METHOD metCreate_S_BV_5 : BOOL
(* S_BV_5*)
IF NOT S_BV_5.xIsCreated THEN
	(* Ziel						UTF8->ASCII						OBJ_NAME_BASE			BacNet Text		Textlistname									BacNet Funktion																BacNet Textlist type												TextId		*)
	S_BV_5._sObjectName		:=	fcUtfToAscii(Standard.CONCAT(	OBJ_NAME_BASE		,	fcGetBcText(	GVL_BACNET.fbBacNetParameter.metGetTextListName(enTypeOfBacNetFunktionIn := enTypeOfBacNetFunktion.Type_Automationsstation,		enTypeOfBacNetTextListIn := enTypeOfBacNetTextList.ENDING		),	'S_BV_5')));
	S_BV_5._sDescription	:= 	fcUtfToAscii(Standard.CONCAT(	OBJ_NAME_DESCRIPTION,	fcGetBcText(	GVL_BACNET.fbBacNetParameter.metGetTextListName(enTypeOfBacNetFunktionIn := enTypeOfBacNetFunktion.Type_Automationsstation,		enTypeOfBacNetTextListIn := enTypeOfBacNetTextList.DESCRIPTION	),	'S_BV_5')));
	(* Create Id from Base Id and Object Nr (Last nummber of Name *)	
	S_BV_5.Create(diInstance := TO_DINT(Standard.CONCAT(TO_STRING(dwOBJ_ID_BASE),'5')));
	(* Check if Created *)
	IF S_BV_5.xIsCreated THEN
		(* Set Group *)
		S_BV_5.setPropertyGroup(WagoTypesBacNet.eBACnetPropertyIdentifier.PROP_PRESENT_VALUE						,WagoTypesBacNet.eBACnetPropertyUpdateGroup.GROUP_CYCLIC);
		S_BV_5.setPropertyGroup(WagoTypesBacNet.eBACnetPropertyIdentifier.PROP_PRIORITY_ARRAY						,WagoTypesBacNet.eBACnetPropertyUpdateGroup.GROUP_CYCLIC);
		S_BV_5.setPropertyGroup(WagoTypesBacNet.eBACnetPropertyIdentifier.PROP_ELAPSED_ACTIVE_TIME					,WagoTypesBacNet.eBACnetPropertyUpdateGroup.GROUP_CYCLIC);
		S_BV_5.setPropertyGroup(WagoTypesBacNet.eBACnetPropertyIdentifier.PROP_DESCRIPTION							,WagoTypesBacNet.eBACnetPropertyUpdateGroup.GROUP_CYCLIC);
		S_BV_5.setPropertyGroup(WagoTypesBacNet.eBACnetPropertyIdentifier.PROP_EVENT_MESSAGE_TEXTS_CONFIG			,WagoTypesBacNet.eBACnetPropertyUpdateGroup.GROUP_CYCLIC);
		(* Set Description to Overwrite retain*)
		S_BV_5.sDescription	:= S_BV_5._sDescription;
		(* Ziel												UTF8->ASCII		BacNet Text		Textlistname									BacNet Funktion																BacNet Textlist type												TextId		*)
		S_BV_5.IEventMessageTextsConfig.sToOffNormal	:=	fcUtfToAscii(	fcGetBcText(	GVL_BACNET.fbBacNetParameter.metGetTextListName(enTypeOfBacNetFunktionIn := enTypeOfBacNetFunktion.Type_Automationsstation,		enTypeOfBacNetTextListIn := enTypeOfBacNetTextList.EVENTMESSAGE	),	'S_BV_5_ToOffNormal'	));		
		S_BV_5.IEventMessageTextsConfig.sToFault		:=	fcUtfToAscii(	fcGetBcText(	GVL_BACNET.fbBacNetParameter.metGetTextListName(enTypeOfBacNetFunktionIn := enTypeOfBacNetFunktion.Type_Automationsstation,		enTypeOfBacNetTextListIn := enTypeOfBacNetTextList.EVENTMESSAGE	),	'S_BV_5_ToFault'		));		
		S_BV_5.IEventMessageTextsConfig.sToNormal		:=	fcUtfToAscii(	fcGetBcText(	GVL_BACNET.fbBacNetParameter.metGetTextListName(enTypeOfBacNetFunktionIn := enTypeOfBacNetFunktion.Type_Automationsstation,		enTypeOfBacNetTextListIn := enTypeOfBacNetTextList.EVENTMESSAGE	),	'S_BV_5_ToNormal'		));		

		(* Ziel												UTF8->ASCII		BacNet Text		Textlistname									BacNet Funktion																BacNet Textlist type												TextId		*)	
		S_BV_5.sActiveText								:= 	fcUtfToAscii(	fcGetBcText(	GVL_BACNET.fbBacNetParameter.metGetTextListName(enTypeOfBacNetFunktionIn := enTypeOfBacNetFunktion.Type_Automationsstation,		enTypeOfBacNetTextListIn := enTypeOfBacNetTextList.PRESENTVALUE	),	'S_BV_5_ST_ACTIVE'		));
		S_BV_5.sInactiveText							:= 	fcUtfToAscii(	fcGetBcText(	GVL_BACNET.fbBacNetParameter.metGetTextListName(enTypeOfBacNetFunktionIn := enTypeOfBacNetFunktion.Type_Automationsstation,		enTypeOfBacNetTextListIn := enTypeOfBacNetTextList.PRESENTVALUE	),	'S_BV_5_ST_INACTIVE'	));	

		(* Ziel												Convert			BacNet Text		Textlistname									BacNet Funktion																	BacNet Textlist type												TextId		*)	
		S_BV_5.udiNotificationClass						:= 	TO_UDINT	(	fcGetBcText(	GVL_BACNET.fbBacNetParameter.metGetTextListName(enTypeOfBacNetFunktionIn := enTypeOfBacNetFunktion.Type_Automationsstation,		enTypeOfBacNetTextListIn := enTypeOfBacNetTextList.NC			),	'S_BV_5_NC'	));	
		S_BV_5.eNotifyType								:= 	WagoTypesBACnet.eBACnetNotifyType.NOTIFY_TYPE_ALARM;		
		S_BV_5.xAlarmValue								:= 	TO_BOOL		(	fcGetBcText(	GVL_BACNET.fbBacNetParameter.metGetTextListName(enTypeOfBacNetFunktionIn := enTypeOfBacNetFunktion.Type_Automationsstation,		enTypeOfBacNetTextListIn := enTypeOfBacNetTextList.NC			),	'S_BV_5_ALV'	));	
		
	ELSE
		S_BV_5.Delete();
	END_IF;
	(* Get Status *)
	metCreate_S_BV_5 := S_BV_5.xIsCreated;	
END_IF;
END_METHOD

METHOD metCreate_I_NC_66 : BOOL

VAR

END_VAR
(* I_NC_66*)
IF NOT I_NC_66.xIsCreated THEN
	(* Ziel						UTF8->ASCII						OBJ_NAME_BASE			BacNet Text		Textlistname									BacNet Funktion																	BacNet Textlist type												TextId		*)
	I_NC_66._sObjectName		:=	fcUtfToAscii(Standard.CONCAT(	OBJ_NAME_BASE		,	fcGetBcText(	GVL_BACNET.fbBacNetParameter.metGetTextListName(enTypeOfBacNetFunktionIn := enTypeOfBacNetFunktion.Type_Automationsstation,		enTypeOfBacNetTextListIn := enTypeOfBacNetTextList.ENDING		),	'I_NC_66')));
	I_NC_66._sDescription	:= 	fcUtfToAscii(Standard.CONCAT(	OBJ_NAME_DESCRIPTION,	fcGetBcText(	GVL_BACNET.fbBacNetParameter.metGetTextListName(enTypeOfBacNetFunktionIn := enTypeOfBacNetFunktion.Type_Automationsstation,		enTypeOfBacNetTextListIn := enTypeOfBacNetTextList.DESCRIPTION	),	'I_NC_66')));
	(* Create Id from Base Id and Object Nr (Last nummber of Name *)	
	I_NC_66.Create(diInstance := 66);
	(* Check if Created *)
	IF I_NC_66.xIsCreated THEN
		(* Set Group *)
		I_NC_66.setPropertyGroup(WagoTypesBacNet.eBACnetPropertyIdentifier.PROP_DESCRIPTION							,WagoTypesBacNet.eBACnetPropertyUpdateGroup.GROUP_CYCLIC);
		
		(* Set Ack Req *)
		I_NC_66.IAckRequired.xToOffNormal	:= TRUE;
		I_NC_66.IAckRequired.xToFault		:= TRUE;
		I_NC_66.IAckRequired.xToNormal		:= FALSE;
		
		(* Ziel												UTF8->ASCII		BacNet Text		Textlistname									BacNet Funktion																	BacNet Textlist type												TextId		*)
		I_NC_66.IEventMessageTextsConfig.sToOffNormal	:=	fcUtfToAscii(	fcGetBcText(	GVL_BACNET.fbBacNetParameter.metGetTextListName(enTypeOfBacNetFunktionIn := enTypeOfBacNetFunktion.Type_Automationsstation,		enTypeOfBacNetTextListIn := enTypeOfBacNetTextList.EVENTMESSAGE	),	'I_NC_66_ToOffNormal'	));		
		I_NC_66.IEventMessageTextsConfig.sToFault		:=	fcUtfToAscii(	fcGetBcText(	GVL_BACNET.fbBacNetParameter.metGetTextListName(enTypeOfBacNetFunktionIn := enTypeOfBacNetFunktion.Type_Automationsstation,		enTypeOfBacNetTextListIn := enTypeOfBacNetTextList.EVENTMESSAGE	),	'I_NC_66_ToFault'		));		
		I_NC_66.IEventMessageTextsConfig.sToNormal		:=	fcUtfToAscii(	fcGetBcText(	GVL_BACNET.fbBacNetParameter.metGetTextListName(enTypeOfBacNetFunktionIn := enTypeOfBacNetFunktion.Type_Automationsstation,		enTypeOfBacNetTextListIn := enTypeOfBacNetTextList.EVENTMESSAGE	),	'I_NC_66_ToNormal'		));		
		
		(* Notification Class & Type *)
		I_NC_66.udiNotificationClass					:=  66;	
		I_NC_66.eNotifyType								:= 	WagoTypesBACnet.eBACnetNotifyType.NOTIFY_TYPE_ALARM;
		(* Ziel												Convert			BacNet Text		Textlistname									BacNet Funktion																	BacNet Textlist type												TextId		*)	
		I_NC_66.IPriority.usiToOffNormal				:= 	TO_USINT(fcUtfToAscii(	fcGetBcText(	GVL_BACNET.fbBacNetParameter.metGetTextListName(enTypeOfBacNetFunktionIn := enTypeOfBacNetFunktion.Type_Automationsstation,		enTypeOfBacNetTextListIn := enTypeOfBacNetTextList.NC	),	'I_NC_66_Prio_ToOffNormal'	)));	
		I_NC_66.IPriority.usiToFault					:= 	TO_USINT(fcUtfToAscii(	fcGetBcText(	GVL_BACNET.fbBacNetParameter.metGetTextListName(enTypeOfBacNetFunktionIn := enTypeOfBacNetFunktion.Type_Automationsstation,		enTypeOfBacNetTextListIn := enTypeOfBacNetTextList.NC	),	'I_NC_66_Prio_ToFault'		)));	
		I_NC_66.IPriority.usiToNormal					:= 	TO_USINT(fcUtfToAscii(	fcGetBcText(	GVL_BACNET.fbBacNetParameter.metGetTextListName(enTypeOfBacNetFunktionIn := enTypeOfBacNetFunktion.Type_Automationsstation,		enTypeOfBacNetTextListIn := enTypeOfBacNetTextList.NC	),	'I_NC_66_Prio_ToNormal'		)));	
		
	ELSE
		I_NC_66.Delete();
	END_IF;
	(* Get Status *)
	metCreate_I_NC_66 := I_NC_66.xIsCreated;	
END_IF;
END_METHOD

METHOD metCreate_J_NC_97 : BOOL

VAR

END_VAR
(* J_NC_97*)
IF NOT J_NC_97.xIsCreated THEN
	(* Ziel						UTF8->ASCII						OBJ_NAME_BASE			BacNet Text		Textlistname									BacNet Funktion																	BacNet Textlist type												TextId		*)
	J_NC_97._sObjectName		:=	fcUtfToAscii(Standard.CONCAT(	OBJ_NAME_BASE		,	fcGetBcText(	GVL_BACNET.fbBacNetParameter.metGetTextListName(enTypeOfBacNetFunktionIn := enTypeOfBacNetFunktion.Type_Automationsstation,		enTypeOfBacNetTextListIn := enTypeOfBacNetTextList.ENDING		),	'J_NC_97')));
	J_NC_97._sDescription	:= 	fcUtfToAscii(Standard.CONCAT(	OBJ_NAME_DESCRIPTION,	fcGetBcText(	GVL_BACNET.fbBacNetParameter.metGetTextListName(enTypeOfBacNetFunktionIn := enTypeOfBacNetFunktion.Type_Automationsstation,		enTypeOfBacNetTextListIn := enTypeOfBacNetTextList.DESCRIPTION	),	'J_NC_97')));
	(* Create Id from Base Id and Object Nr (Last nummber of Name *)	
	J_NC_97.Create(diInstance := 97);
	(* Check if Created *)
	IF J_NC_97.xIsCreated THEN
		(* Set Group *)
		J_NC_97.setPropertyGroup(WagoTypesBacNet.eBACnetPropertyIdentifier.PROP_DESCRIPTION							,WagoTypesBacNet.eBACnetPropertyUpdateGroup.GROUP_CYCLIC);
		
		(* Set Ack Req *)
		J_NC_97.IAckRequired.xToOffNormal	:= FALSE;
		J_NC_97.IAckRequired.xToFault		:= TRUE;
		J_NC_97.IAckRequired.xToNormal		:= FALSE;
		
		(* Ziel												UTF8->ASCII		BacNet Text		Textlistname									BacNet Funktion																	BacNet Textlist type												TextId		*)
		J_NC_97.IEventMessageTextsConfig.sToOffNormal	:=	fcUtfToAscii(	fcGetBcText(	GVL_BACNET.fbBacNetParameter.metGetTextListName(enTypeOfBacNetFunktionIn := enTypeOfBacNetFunktion.Type_Automationsstation,		enTypeOfBacNetTextListIn := enTypeOfBacNetTextList.EVENTMESSAGE	),	'J_NC_97_ToOffNormal'	));		
		J_NC_97.IEventMessageTextsConfig.sToFault		:=	fcUtfToAscii(	fcGetBcText(	GVL_BACNET.fbBacNetParameter.metGetTextListName(enTypeOfBacNetFunktionIn := enTypeOfBacNetFunktion.Type_Automationsstation,		enTypeOfBacNetTextListIn := enTypeOfBacNetTextList.EVENTMESSAGE	),	'J_NC_97_ToFault'		));		
		J_NC_97.IEventMessageTextsConfig.sToNormal		:=	fcUtfToAscii(	fcGetBcText(	GVL_BACNET.fbBacNetParameter.metGetTextListName(enTypeOfBacNetFunktionIn := enTypeOfBacNetFunktion.Type_Automationsstation,		enTypeOfBacNetTextListIn := enTypeOfBacNetTextList.EVENTMESSAGE	),	'J_NC_97_ToNormal'		));		
		
		(* Notification Class & Type *)
		J_NC_97.udiNotificationClass					:=  97;	
		J_NC_97.eNotifyType								:= 	WagoTypesBACnet.eBACnetNotifyType.NOTIFY_TYPE_ALARM;
		(* Ziel												Convert			BacNet Text		Textlistname									BacNet Funktion																	BacNet Textlist type												TextId		*)	
		J_NC_97.IPriority.usiToOffNormal				:= 	TO_USINT(fcUtfToAscii(	fcGetBcText(	GVL_BACNET.fbBacNetParameter.metGetTextListName(enTypeOfBacNetFunktionIn := enTypeOfBacNetFunktion.Type_Automationsstation,		enTypeOfBacNetTextListIn := enTypeOfBacNetTextList.NC	),	'J_NC_97_Prio_ToOffNormal'	)));	
		J_NC_97.IPriority.usiToFault					:= 	TO_USINT(fcUtfToAscii(	fcGetBcText(	GVL_BACNET.fbBacNetParameter.metGetTextListName(enTypeOfBacNetFunktionIn := enTypeOfBacNetFunktion.Type_Automationsstation,		enTypeOfBacNetTextListIn := enTypeOfBacNetTextList.NC	),	'J_NC_97_Prio_ToFault'		)));	
		J_NC_97.IPriority.usiToNormal					:= 	TO_USINT(fcUtfToAscii(	fcGetBcText(	GVL_BACNET.fbBacNetParameter.metGetTextListName(enTypeOfBacNetFunktionIn := enTypeOfBacNetFunktion.Type_Automationsstation,		enTypeOfBacNetTextListIn := enTypeOfBacNetTextList.NC	),	'J_NC_97_Prio_ToNormal'		)));	
		
	ELSE
		J_NC_97.Delete();
	END_IF;
	(* Get Status *)
	metCreate_J_NC_97 := J_NC_97.xIsCreated;	
END_IF;
END_METHOD

METHOD metCreate_J_NC_98 : BOOL

VAR

END_VAR
(* J_NC_98*)
IF NOT J_NC_98.xIsCreated THEN
	(* Ziel						UTF8->ASCII						OBJ_NAME_BASE			BacNet Text		Textlistname									BacNet Funktion																	BacNet Textlist type												TextId		*)
	J_NC_98._sObjectName		:=	fcUtfToAscii(Standard.CONCAT(	OBJ_NAME_BASE		,	fcGetBcText(	GVL_BACNET.fbBacNetParameter.metGetTextListName(enTypeOfBacNetFunktionIn := enTypeOfBacNetFunktion.Type_Automationsstation,		enTypeOfBacNetTextListIn := enTypeOfBacNetTextList.ENDING		),	'J_NC_98')));
	J_NC_98._sDescription	:= 	fcUtfToAscii(Standard.CONCAT(	OBJ_NAME_DESCRIPTION,	fcGetBcText(	GVL_BACNET.fbBacNetParameter.metGetTextListName(enTypeOfBacNetFunktionIn := enTypeOfBacNetFunktion.Type_Automationsstation,		enTypeOfBacNetTextListIn := enTypeOfBacNetTextList.DESCRIPTION	),	'J_NC_98')));
	(* Create Id from Base Id and Object Nr (Last nummber of Name *)	
	J_NC_98.Create(diInstance := 98);
	(* Check if Created *)
	IF J_NC_98.xIsCreated THEN
		(* Set Group *)
		J_NC_98.setPropertyGroup(WagoTypesBacNet.eBACnetPropertyIdentifier.PROP_DESCRIPTION							,WagoTypesBacNet.eBACnetPropertyUpdateGroup.GROUP_CYCLIC);
		
		(* Set Ack Req *)
		J_NC_98.IAckRequired.xToOffNormal	:= TRUE;
		J_NC_98.IAckRequired.xToFault		:= TRUE;
		J_NC_98.IAckRequired.xToNormal		:= FALSE;
		
		(* Ziel												UTF8->ASCII		BacNet Text		Textlistname									BacNet Funktion																	BacNet Textlist type												TextId		*)
		J_NC_98.IEventMessageTextsConfig.sToOffNormal	:=	fcUtfToAscii(	fcGetBcText(	GVL_BACNET.fbBacNetParameter.metGetTextListName(enTypeOfBacNetFunktionIn := enTypeOfBacNetFunktion.Type_Automationsstation,		enTypeOfBacNetTextListIn := enTypeOfBacNetTextList.EVENTMESSAGE	),	'J_NC_98_ToOffNormal'	));		
		J_NC_98.IEventMessageTextsConfig.sToFault		:=	fcUtfToAscii(	fcGetBcText(	GVL_BACNET.fbBacNetParameter.metGetTextListName(enTypeOfBacNetFunktionIn := enTypeOfBacNetFunktion.Type_Automationsstation,		enTypeOfBacNetTextListIn := enTypeOfBacNetTextList.EVENTMESSAGE	),	'J_NC_98_ToFault'		));		
		J_NC_98.IEventMessageTextsConfig.sToNormal		:=	fcUtfToAscii(	fcGetBcText(	GVL_BACNET.fbBacNetParameter.metGetTextListName(enTypeOfBacNetFunktionIn := enTypeOfBacNetFunktion.Type_Automationsstation,		enTypeOfBacNetTextListIn := enTypeOfBacNetTextList.EVENTMESSAGE	),	'J_NC_98_ToNormal'		));		
		
		(* Notification Class & Type *)
		J_NC_98.udiNotificationClass					:=  98;	
		J_NC_98.eNotifyType								:= 	WagoTypesBACnet.eBACnetNotifyType.NOTIFY_TYPE_ALARM;
		(* Ziel												Convert			BacNet Text		Textlistname									BacNet Funktion																	BacNet Textlist type												TextId		*)	
		J_NC_98.IPriority.usiToOffNormal				:= 	TO_USINT(fcUtfToAscii(	fcGetBcText(	GVL_BACNET.fbBacNetParameter.metGetTextListName(enTypeOfBacNetFunktionIn := enTypeOfBacNetFunktion.Type_Automationsstation,		enTypeOfBacNetTextListIn := enTypeOfBacNetTextList.NC	),	'J_NC_98_Prio_ToOffNormal'	)));	
		J_NC_98.IPriority.usiToFault					:= 	TO_USINT(fcUtfToAscii(	fcGetBcText(	GVL_BACNET.fbBacNetParameter.metGetTextListName(enTypeOfBacNetFunktionIn := enTypeOfBacNetFunktion.Type_Automationsstation,		enTypeOfBacNetTextListIn := enTypeOfBacNetTextList.NC	),	'J_NC_98_Prio_ToFault'		)));	
		J_NC_98.IPriority.usiToNormal					:= 	TO_USINT(fcUtfToAscii(	fcGetBcText(	GVL_BACNET.fbBacNetParameter.metGetTextListName(enTypeOfBacNetFunktionIn := enTypeOfBacNetFunktion.Type_Automationsstation,		enTypeOfBacNetTextListIn := enTypeOfBacNetTextList.NC	),	'J_NC_98_Prio_ToNormal'		)));	
		
	ELSE
		J_NC_98.Delete();
	END_IF;
	(* Get Status *)
	metCreate_J_NC_98 := J_NC_98.xIsCreated;	
END_IF;
END_METHOD

METHOD metCreate_J_NC_99 : BOOL

VAR

END_VAR
(* J_NC_99*)
IF NOT J_NC_99.xIsCreated THEN
	(* Ziel						UTF8->ASCII						OBJ_NAME_BASE			BacNet Text		Textlistname									BacNet Funktion																	BacNet Textlist type												TextId		*)
	J_NC_99._sObjectName		:=	fcUtfToAscii(Standard.CONCAT(	OBJ_NAME_BASE		,	fcGetBcText(	GVL_BACNET.fbBacNetParameter.metGetTextListName(enTypeOfBacNetFunktionIn := enTypeOfBacNetFunktion.Type_Automationsstation,		enTypeOfBacNetTextListIn := enTypeOfBacNetTextList.ENDING		),	'J_NC_99')));
	J_NC_99._sDescription	:= 	fcUtfToAscii(Standard.CONCAT(	OBJ_NAME_DESCRIPTION,	fcGetBcText(	GVL_BACNET.fbBacNetParameter.metGetTextListName(enTypeOfBacNetFunktionIn := enTypeOfBacNetFunktion.Type_Automationsstation,		enTypeOfBacNetTextListIn := enTypeOfBacNetTextList.DESCRIPTION	),	'J_NC_99')));
	(* Create Id from Base Id and Object Nr (Last nummber of Name *)	
	J_NC_99.Create(diInstance := 99);
	(* Check if Created *)
	IF J_NC_99.xIsCreated THEN
		(* Set Group *)
		J_NC_99.setPropertyGroup(WagoTypesBacNet.eBACnetPropertyIdentifier.PROP_DESCRIPTION							,WagoTypesBacNet.eBACnetPropertyUpdateGroup.GROUP_CYCLIC);
		
		(* Set Ack Req *)
		J_NC_99.IAckRequired.xToOffNormal	:= TRUE;
		J_NC_99.IAckRequired.xToFault		:= TRUE;
		J_NC_99.IAckRequired.xToNormal		:= TRUE;
		
		(* Ziel												UTF8->ASCII		BacNet Text		Textlistname									BacNet Funktion																	BacNet Textlist type												TextId		*)
		J_NC_99.IEventMessageTextsConfig.sToOffNormal	:=	fcUtfToAscii(	fcGetBcText(	GVL_BACNET.fbBacNetParameter.metGetTextListName(enTypeOfBacNetFunktionIn := enTypeOfBacNetFunktion.Type_Automationsstation,		enTypeOfBacNetTextListIn := enTypeOfBacNetTextList.EVENTMESSAGE	),	'J_NC_99_ToOffNormal'	));		
		J_NC_99.IEventMessageTextsConfig.sToFault		:=	fcUtfToAscii(	fcGetBcText(	GVL_BACNET.fbBacNetParameter.metGetTextListName(enTypeOfBacNetFunktionIn := enTypeOfBacNetFunktion.Type_Automationsstation,		enTypeOfBacNetTextListIn := enTypeOfBacNetTextList.EVENTMESSAGE	),	'J_NC_99_ToFault'		));		
		J_NC_99.IEventMessageTextsConfig.sToNormal		:=	fcUtfToAscii(	fcGetBcText(	GVL_BACNET.fbBacNetParameter.metGetTextListName(enTypeOfBacNetFunktionIn := enTypeOfBacNetFunktion.Type_Automationsstation,		enTypeOfBacNetTextListIn := enTypeOfBacNetTextList.EVENTMESSAGE	),	'J_NC_99_ToNormal'		));		
		
		(* Notification Class & Type *)
		J_NC_99.udiNotificationClass					:=  99;	
		J_NC_99.eNotifyType								:= 	WagoTypesBACnet.eBACnetNotifyType.NOTIFY_TYPE_ALARM;
		(* Ziel												Convert			BacNet Text		Textlistname									BacNet Funktion																	BacNet Textlist type												TextId		*)	
		J_NC_99.IPriority.usiToOffNormal				:= 	TO_USINT(fcUtfToAscii(	fcGetBcText(	GVL_BACNET.fbBacNetParameter.metGetTextListName(enTypeOfBacNetFunktionIn := enTypeOfBacNetFunktion.Type_Automationsstation,		enTypeOfBacNetTextListIn := enTypeOfBacNetTextList.NC	),	'J_NC_99_Prio_ToOffNormal'	)));	
		J_NC_99.IPriority.usiToFault					:= 	TO_USINT(fcUtfToAscii(	fcGetBcText(	GVL_BACNET.fbBacNetParameter.metGetTextListName(enTypeOfBacNetFunktionIn := enTypeOfBacNetFunktion.Type_Automationsstation,		enTypeOfBacNetTextListIn := enTypeOfBacNetTextList.NC	),	'J_NC_99_Prio_ToFault'		)));	
		J_NC_99.IPriority.usiToNormal					:= 	TO_USINT(fcUtfToAscii(	fcGetBcText(	GVL_BACNET.fbBacNetParameter.metGetTextListName(enTypeOfBacNetFunktionIn := enTypeOfBacNetFunktion.Type_Automationsstation,		enTypeOfBacNetTextListIn := enTypeOfBacNetTextList.NC	),	'J_NC_99_Prio_ToNormal'		)));	
		
	ELSE
		J_NC_99.Delete();
	END_IF;
	(* Get Status *)
	metCreate_J_NC_99 := J_NC_99.xIsCreated;	
END_IF;
END_METHOD

METHOD metCreate_K_NC_128 : BOOL

VAR

END_VAR
(* K_NC_128*)
IF NOT K_NC_128.xIsCreated THEN
	(* Ziel						UTF8->ASCII						OBJ_NAME_BASE			BacNet Text		Textlistname									BacNet Funktion																	BacNet Textlist type												TextId		*)
	K_NC_128._sObjectName		:=	fcUtfToAscii(Standard.CONCAT(	OBJ_NAME_BASE		,	fcGetBcText(	GVL_BACNET.fbBacNetParameter.metGetTextListName(enTypeOfBacNetFunktionIn := enTypeOfBacNetFunktion.Type_Automationsstation,		enTypeOfBacNetTextListIn := enTypeOfBacNetTextList.ENDING		),	'K_NC_128')));
	K_NC_128._sDescription	:= 	fcUtfToAscii(Standard.CONCAT(	OBJ_NAME_DESCRIPTION,	fcGetBcText(	GVL_BACNET.fbBacNetParameter.metGetTextListName(enTypeOfBacNetFunktionIn := enTypeOfBacNetFunktion.Type_Automationsstation,		enTypeOfBacNetTextListIn := enTypeOfBacNetTextList.DESCRIPTION	),	'K_NC_128')));
	(* Create Id from Base Id and Object Nr (Last nummber of Name *)	
	K_NC_128.Create(diInstance := 128);
	(* Check if Created *)
	IF K_NC_128.xIsCreated THEN
		(* Set Group *)
		K_NC_128.setPropertyGroup(WagoTypesBacNet.eBACnetPropertyIdentifier.PROP_DESCRIPTION							,WagoTypesBacNet.eBACnetPropertyUpdateGroup.GROUP_CYCLIC);
		
		(* Set Ack Req *)
		K_NC_128.IAckRequired.xToOffNormal	:= FALSE;
		K_NC_128.IAckRequired.xToFault		:= FALSE;
		K_NC_128.IAckRequired.xToNormal		:= FALSE;
		
		(* Ziel												UTF8->ASCII		BacNet Text		Textlistname									BacNet Funktion																	BacNet Textlist type												TextId		*)
		K_NC_128.IEventMessageTextsConfig.sToOffNormal	:=	fcUtfToAscii(	fcGetBcText(	GVL_BACNET.fbBacNetParameter.metGetTextListName(enTypeOfBacNetFunktionIn := enTypeOfBacNetFunktion.Type_Automationsstation,		enTypeOfBacNetTextListIn := enTypeOfBacNetTextList.EVENTMESSAGE	),	'K_NC_128_ToOffNormal'	));		
		K_NC_128.IEventMessageTextsConfig.sToFault		:=	fcUtfToAscii(	fcGetBcText(	GVL_BACNET.fbBacNetParameter.metGetTextListName(enTypeOfBacNetFunktionIn := enTypeOfBacNetFunktion.Type_Automationsstation,		enTypeOfBacNetTextListIn := enTypeOfBacNetTextList.EVENTMESSAGE	),	'K_NC_128_ToFault'		));		
		K_NC_128.IEventMessageTextsConfig.sToNormal		:=	fcUtfToAscii(	fcGetBcText(	GVL_BACNET.fbBacNetParameter.metGetTextListName(enTypeOfBacNetFunktionIn := enTypeOfBacNetFunktion.Type_Automationsstation,		enTypeOfBacNetTextListIn := enTypeOfBacNetTextList.EVENTMESSAGE	),	'K_NC_128_ToNormal'		));		
		
		(* Notification Class & Type *)
		K_NC_128.udiNotificationClass					:=  128;	
		K_NC_128.eNotifyType								:= 	WagoTypesBACnet.eBACnetNotifyType.NOTIFY_TYPE_ALARM;
		(* Ziel												Convert			BacNet Text		Textlistname									BacNet Funktion																	BacNet Textlist type												TextId		*)	
		K_NC_128.IPriority.usiToOffNormal				:= 	TO_USINT(fcUtfToAscii(	fcGetBcText(	GVL_BACNET.fbBacNetParameter.metGetTextListName(enTypeOfBacNetFunktionIn := enTypeOfBacNetFunktion.Type_Automationsstation,		enTypeOfBacNetTextListIn := enTypeOfBacNetTextList.NC	),	'K_NC_128_Prio_ToOffNormal'	)));	
		K_NC_128.IPriority.usiToFault					:= 	TO_USINT(fcUtfToAscii(	fcGetBcText(	GVL_BACNET.fbBacNetParameter.metGetTextListName(enTypeOfBacNetFunktionIn := enTypeOfBacNetFunktion.Type_Automationsstation,		enTypeOfBacNetTextListIn := enTypeOfBacNetTextList.NC	),	'K_NC_128_Prio_ToFault'		)));	
		K_NC_128.IPriority.usiToNormal					:= 	TO_USINT(fcUtfToAscii(	fcGetBcText(	GVL_BACNET.fbBacNetParameter.metGetTextListName(enTypeOfBacNetFunktionIn := enTypeOfBacNetFunktion.Type_Automationsstation,		enTypeOfBacNetTextListIn := enTypeOfBacNetTextList.NC	),	'K_NC_128_Prio_ToNormal'		)));	
		
	ELSE
		K_NC_128.Delete();
	END_IF;
	(* Get Status *)
	metCreate_K_NC_128 := K_NC_128.xIsCreated;	
END_IF;
END_METHOD

METHOD metCreate_H_NC_35 : BOOL

VAR

END_VAR
(* H_NC_35*)
IF NOT H_NC_35.xIsCreated THEN
	(* Ziel						UTF8->ASCII						OBJ_NAME_BASE			BacNet Text		Textlistname									BacNet Funktion																	BacNet Textlist type												TextId		*)
	H_NC_35._sObjectName		:=	fcUtfToAscii(Standard.CONCAT(	OBJ_NAME_BASE		,	fcGetBcText(	GVL_BACNET.fbBacNetParameter.metGetTextListName(enTypeOfBacNetFunktionIn := enTypeOfBacNetFunktion.Type_Automationsstation,		enTypeOfBacNetTextListIn := enTypeOfBacNetTextList.ENDING		),	'H_NC_35')));
	H_NC_35._sDescription	:= 	fcUtfToAscii(Standard.CONCAT(	OBJ_NAME_DESCRIPTION,	fcGetBcText(	GVL_BACNET.fbBacNetParameter.metGetTextListName(enTypeOfBacNetFunktionIn := enTypeOfBacNetFunktion.Type_Automationsstation,		enTypeOfBacNetTextListIn := enTypeOfBacNetTextList.DESCRIPTION	),	'H_NC_35')));
	(* Create Id from Base Id and Object Nr (Last nummber of Name *)	
	H_NC_35.Create(diInstance := 35);
	(* Check if Created *)
	IF H_NC_35.xIsCreated THEN
		(* Set Group *)
		H_NC_35.setPropertyGroup(WagoTypesBacNet.eBACnetPropertyIdentifier.PROP_DESCRIPTION							,WagoTypesBacNet.eBACnetPropertyUpdateGroup.GROUP_CYCLIC);
		
		(* Set Ack Req *)
		H_NC_35.IAckRequired.xToOffNormal	:= TRUE;
		H_NC_35.IAckRequired.xToFault		:= TRUE;
		H_NC_35.IAckRequired.xToNormal		:= TRUE;
		
		(* Ziel												UTF8->ASCII		BacNet Text		Textlistname									BacNet Funktion																	BacNet Textlist type												TextId		*)
		H_NC_35.IEventMessageTextsConfig.sToOffNormal	:=	fcUtfToAscii(	fcGetBcText(	GVL_BACNET.fbBacNetParameter.metGetTextListName(enTypeOfBacNetFunktionIn := enTypeOfBacNetFunktion.Type_Automationsstation,		enTypeOfBacNetTextListIn := enTypeOfBacNetTextList.EVENTMESSAGE	),	'H_NC_35_ToOffNormal'	));		
		H_NC_35.IEventMessageTextsConfig.sToFault		:=	fcUtfToAscii(	fcGetBcText(	GVL_BACNET.fbBacNetParameter.metGetTextListName(enTypeOfBacNetFunktionIn := enTypeOfBacNetFunktion.Type_Automationsstation,		enTypeOfBacNetTextListIn := enTypeOfBacNetTextList.EVENTMESSAGE	),	'H_NC_35_ToFault'		));		
		H_NC_35.IEventMessageTextsConfig.sToNormal		:=	fcUtfToAscii(	fcGetBcText(	GVL_BACNET.fbBacNetParameter.metGetTextListName(enTypeOfBacNetFunktionIn := enTypeOfBacNetFunktion.Type_Automationsstation,		enTypeOfBacNetTextListIn := enTypeOfBacNetTextList.EVENTMESSAGE	),	'H_NC_35_ToNormal'		));		
		
		(* Notification Class & Type *)
		H_NC_35.udiNotificationClass					:=  35;	
		H_NC_35.eNotifyType								:= 	WagoTypesBACnet.eBACnetNotifyType.NOTIFY_TYPE_ALARM;
		(* Ziel												Convert			BacNet Text		Textlistname									BacNet Funktion																	BacNet Textlist type												TextId		*)	
		H_NC_35.IPriority.usiToOffNormal				:= 	TO_USINT(fcUtfToAscii(	fcGetBcText(	GVL_BACNET.fbBacNetParameter.metGetTextListName(enTypeOfBacNetFunktionIn := enTypeOfBacNetFunktion.Type_Automationsstation,		enTypeOfBacNetTextListIn := enTypeOfBacNetTextList.NC	),	'H_NC_35_Prio_ToOffNormal'	)));	
		H_NC_35.IPriority.usiToFault					:= 	TO_USINT(fcUtfToAscii(	fcGetBcText(	GVL_BACNET.fbBacNetParameter.metGetTextListName(enTypeOfBacNetFunktionIn := enTypeOfBacNetFunktion.Type_Automationsstation,		enTypeOfBacNetTextListIn := enTypeOfBacNetTextList.NC	),	'H_NC_35_Prio_ToFault'		)));	
		H_NC_35.IPriority.usiToNormal					:= 	TO_USINT(fcUtfToAscii(	fcGetBcText(	GVL_BACNET.fbBacNetParameter.metGetTextListName(enTypeOfBacNetFunktionIn := enTypeOfBacNetFunktion.Type_Automationsstation,		enTypeOfBacNetTextListIn := enTypeOfBacNetTextList.NC	),	'H_NC_35_Prio_ToNormal'		)));	
		
	ELSE
		H_NC_35.Delete();
	END_IF;
	(* Get Status *)
	metCreate_H_NC_35 := H_NC_35.xIsCreated;	
END_IF;
END_METHOD

METHOD metCreate_I_NC_64 : BOOL

VAR

END_VAR
(* I_NC_64*)
IF NOT I_NC_64.xIsCreated THEN
	(* Ziel						UTF8->ASCII						OBJ_NAME_BASE			BacNet Text		Textlistname									BacNet Funktion																	BacNet Textlist type												TextId		*)
	I_NC_64._sObjectName		:=	fcUtfToAscii(Standard.CONCAT(	OBJ_NAME_BASE		,	fcGetBcText(	GVL_BACNET.fbBacNetParameter.metGetTextListName(enTypeOfBacNetFunktionIn := enTypeOfBacNetFunktion.Type_Automationsstation,		enTypeOfBacNetTextListIn := enTypeOfBacNetTextList.ENDING		),	'I_NC_64')));
	I_NC_64._sDescription	:= 	fcUtfToAscii(Standard.CONCAT(	OBJ_NAME_DESCRIPTION,	fcGetBcText(	GVL_BACNET.fbBacNetParameter.metGetTextListName(enTypeOfBacNetFunktionIn := enTypeOfBacNetFunktion.Type_Automationsstation,		enTypeOfBacNetTextListIn := enTypeOfBacNetTextList.DESCRIPTION	),	'I_NC_64')));
	(* Create Id from Base Id and Object Nr (Last nummber of Name *)	
	I_NC_64.Create(diInstance := 64);
	(* Check if Created *)
	IF I_NC_64.xIsCreated THEN
		(* Set Group *)
		I_NC_64.setPropertyGroup(WagoTypesBacNet.eBACnetPropertyIdentifier.PROP_DESCRIPTION							,WagoTypesBacNet.eBACnetPropertyUpdateGroup.GROUP_CYCLIC);
		
		(* Set Ack Req *)
		I_NC_64.IAckRequired.xToOffNormal	:= FALSE;
		I_NC_64.IAckRequired.xToFault		:= FALSE;
		I_NC_64.IAckRequired.xToNormal		:= FALSE;
		
		(* Ziel												UTF8->ASCII		BacNet Text		Textlistname									BacNet Funktion																	BacNet Textlist type												TextId		*)
		I_NC_64.IEventMessageTextsConfig.sToOffNormal	:=	fcUtfToAscii(	fcGetBcText(	GVL_BACNET.fbBacNetParameter.metGetTextListName(enTypeOfBacNetFunktionIn := enTypeOfBacNetFunktion.Type_Automationsstation,		enTypeOfBacNetTextListIn := enTypeOfBacNetTextList.EVENTMESSAGE	),	'I_NC_64_ToOffNormal'	));		
		I_NC_64.IEventMessageTextsConfig.sToFault		:=	fcUtfToAscii(	fcGetBcText(	GVL_BACNET.fbBacNetParameter.metGetTextListName(enTypeOfBacNetFunktionIn := enTypeOfBacNetFunktion.Type_Automationsstation,		enTypeOfBacNetTextListIn := enTypeOfBacNetTextList.EVENTMESSAGE	),	'I_NC_64_ToFault'		));		
		I_NC_64.IEventMessageTextsConfig.sToNormal		:=	fcUtfToAscii(	fcGetBcText(	GVL_BACNET.fbBacNetParameter.metGetTextListName(enTypeOfBacNetFunktionIn := enTypeOfBacNetFunktion.Type_Automationsstation,		enTypeOfBacNetTextListIn := enTypeOfBacNetTextList.EVENTMESSAGE	),	'I_NC_64_ToNormal'		));		
		
		(* Notification Class & Type *)
		I_NC_64.udiNotificationClass					:=  64;	
		I_NC_64.eNotifyType								:= 	WagoTypesBACnet.eBACnetNotifyType.NOTIFY_TYPE_ALARM;
		(* Ziel												Convert			BacNet Text		Textlistname									BacNet Funktion																	BacNet Textlist type												TextId		*)	
		I_NC_64.IPriority.usiToOffNormal				:= 	TO_USINT(fcUtfToAscii(	fcGetBcText(	GVL_BACNET.fbBacNetParameter.metGetTextListName(enTypeOfBacNetFunktionIn := enTypeOfBacNetFunktion.Type_Automationsstation,		enTypeOfBacNetTextListIn := enTypeOfBacNetTextList.NC	),	'I_NC_64_Prio_ToOffNormal'	)));	
		I_NC_64.IPriority.usiToFault					:= 	TO_USINT(fcUtfToAscii(	fcGetBcText(	GVL_BACNET.fbBacNetParameter.metGetTextListName(enTypeOfBacNetFunktionIn := enTypeOfBacNetFunktion.Type_Automationsstation,		enTypeOfBacNetTextListIn := enTypeOfBacNetTextList.NC	),	'I_NC_64_Prio_ToFault'		)));	
		I_NC_64.IPriority.usiToNormal					:= 	TO_USINT(fcUtfToAscii(	fcGetBcText(	GVL_BACNET.fbBacNetParameter.metGetTextListName(enTypeOfBacNetFunktionIn := enTypeOfBacNetFunktion.Type_Automationsstation,		enTypeOfBacNetTextListIn := enTypeOfBacNetTextList.NC	),	'I_NC_64_Prio_ToNormal'		)));	
		
	ELSE
		I_NC_64.Delete();
	END_IF;
	(* Get Status *)
	metCreate_I_NC_64 := I_NC_64.xIsCreated;	
END_IF;
END_METHOD

METHOD metCreate_I_NC_67 : BOOL

VAR

END_VAR
(* I_NC_67*)
IF NOT I_NC_67.xIsCreated THEN
	(* Ziel						UTF8->ASCII						OBJ_NAME_BASE			BacNet Text		Textlistname									BacNet Funktion																	BacNet Textlist type												TextId		*)
	I_NC_67._sObjectName		:=	fcUtfToAscii(Standard.CONCAT(	OBJ_NAME_BASE		,	fcGetBcText(	GVL_BACNET.fbBacNetParameter.metGetTextListName(enTypeOfBacNetFunktionIn := enTypeOfBacNetFunktion.Type_Automationsstation,		enTypeOfBacNetTextListIn := enTypeOfBacNetTextList.ENDING		),	'I_NC_67')));
	I_NC_67._sDescription	:= 	fcUtfToAscii(Standard.CONCAT(	OBJ_NAME_DESCRIPTION,	fcGetBcText(	GVL_BACNET.fbBacNetParameter.metGetTextListName(enTypeOfBacNetFunktionIn := enTypeOfBacNetFunktion.Type_Automationsstation,		enTypeOfBacNetTextListIn := enTypeOfBacNetTextList.DESCRIPTION	),	'I_NC_67')));
	(* Create Id from Base Id and Object Nr (Last nummber of Name *)	
	I_NC_67.Create(diInstance := 67);
	(* Check if Created *)
	IF I_NC_67.xIsCreated THEN
		(* Set Group *)
		I_NC_67.setPropertyGroup(WagoTypesBacNet.eBACnetPropertyIdentifier.PROP_DESCRIPTION							,WagoTypesBacNet.eBACnetPropertyUpdateGroup.GROUP_CYCLIC);
		
		(* Set Ack Req *)
		I_NC_67.IAckRequired.xToOffNormal	:= TRUE;
		I_NC_67.IAckRequired.xToFault		:= TRUE;
		I_NC_67.IAckRequired.xToNormal		:= TRUE;
		
		(* Ziel												UTF8->ASCII		BacNet Text		Textlistname									BacNet Funktion																	BacNet Textlist type												TextId		*)
		I_NC_67.IEventMessageTextsConfig.sToOffNormal	:=	fcUtfToAscii(	fcGetBcText(	GVL_BACNET.fbBacNetParameter.metGetTextListName(enTypeOfBacNetFunktionIn := enTypeOfBacNetFunktion.Type_Automationsstation,		enTypeOfBacNetTextListIn := enTypeOfBacNetTextList.EVENTMESSAGE	),	'I_NC_67_ToOffNormal'	));		
		I_NC_67.IEventMessageTextsConfig.sToFault		:=	fcUtfToAscii(	fcGetBcText(	GVL_BACNET.fbBacNetParameter.metGetTextListName(enTypeOfBacNetFunktionIn := enTypeOfBacNetFunktion.Type_Automationsstation,		enTypeOfBacNetTextListIn := enTypeOfBacNetTextList.EVENTMESSAGE	),	'I_NC_67_ToFault'		));		
		I_NC_67.IEventMessageTextsConfig.sToNormal		:=	fcUtfToAscii(	fcGetBcText(	GVL_BACNET.fbBacNetParameter.metGetTextListName(enTypeOfBacNetFunktionIn := enTypeOfBacNetFunktion.Type_Automationsstation,		enTypeOfBacNetTextListIn := enTypeOfBacNetTextList.EVENTMESSAGE	),	'I_NC_67_ToNormal'		));		
		
		(* Notification Class & Type *)
		I_NC_67.udiNotificationClass					:=  67;	
		I_NC_67.eNotifyType								:= 	WagoTypesBACnet.eBACnetNotifyType.NOTIFY_TYPE_ALARM;
		(* Ziel												Convert			BacNet Text		Textlistname									BacNet Funktion																	BacNet Textlist type												TextId		*)	
		I_NC_67.IPriority.usiToOffNormal				:= 	TO_USINT(fcUtfToAscii(	fcGetBcText(	GVL_BACNET.fbBacNetParameter.metGetTextListName(enTypeOfBacNetFunktionIn := enTypeOfBacNetFunktion.Type_Automationsstation,		enTypeOfBacNetTextListIn := enTypeOfBacNetTextList.NC	),	'I_NC_67_Prio_ToOffNormal'	)));	
		I_NC_67.IPriority.usiToFault					:= 	TO_USINT(fcUtfToAscii(	fcGetBcText(	GVL_BACNET.fbBacNetParameter.metGetTextListName(enTypeOfBacNetFunktionIn := enTypeOfBacNetFunktion.Type_Automationsstation,		enTypeOfBacNetTextListIn := enTypeOfBacNetTextList.NC	),	'I_NC_67_Prio_ToFault'		)));	
		I_NC_67.IPriority.usiToNormal					:= 	TO_USINT(fcUtfToAscii(	fcGetBcText(	GVL_BACNET.fbBacNetParameter.metGetTextListName(enTypeOfBacNetFunktionIn := enTypeOfBacNetFunktion.Type_Automationsstation,		enTypeOfBacNetTextListIn := enTypeOfBacNetTextList.NC	),	'I_NC_67_Prio_ToNormal'		)));	
		
	ELSE
		I_NC_67.Delete();
	END_IF;
	(* Get Status *)
	metCreate_I_NC_67 := I_NC_67.xIsCreated;	
END_IF;
END_METHOD

METHOD metCreate_J_NC_96 : BOOL

VAR

END_VAR
(* J_NC_96*)
IF NOT J_NC_96.xIsCreated THEN
	(* Ziel						UTF8->ASCII						OBJ_NAME_BASE			BacNet Text		Textlistname									BacNet Funktion																	BacNet Textlist type												TextId		*)
	J_NC_96._sObjectName		:=	fcUtfToAscii(Standard.CONCAT(	OBJ_NAME_BASE		,	fcGetBcText(	GVL_BACNET.fbBacNetParameter.metGetTextListName(enTypeOfBacNetFunktionIn := enTypeOfBacNetFunktion.Type_Automationsstation,		enTypeOfBacNetTextListIn := enTypeOfBacNetTextList.ENDING		),	'J_NC_96')));
	J_NC_96._sDescription	:= 	fcUtfToAscii(Standard.CONCAT(	OBJ_NAME_DESCRIPTION,	fcGetBcText(	GVL_BACNET.fbBacNetParameter.metGetTextListName(enTypeOfBacNetFunktionIn := enTypeOfBacNetFunktion.Type_Automationsstation,		enTypeOfBacNetTextListIn := enTypeOfBacNetTextList.DESCRIPTION	),	'J_NC_96')));
	(* Create Id from Base Id and Object Nr (Last nummber of Name *)	
	J_NC_96.Create(diInstance := 96);
	(* Check if Created *)
	IF J_NC_96.xIsCreated THEN
		(* Set Group *)
		J_NC_96.setPropertyGroup(WagoTypesBacNet.eBACnetPropertyIdentifier.PROP_DESCRIPTION							,WagoTypesBacNet.eBACnetPropertyUpdateGroup.GROUP_CYCLIC);
		
		(* Set Ack Req *)
		J_NC_96.IAckRequired.xToOffNormal	:= FALSE;
		J_NC_96.IAckRequired.xToFault		:= FALSE;
		J_NC_96.IAckRequired.xToNormal		:= FALSE;
		
		(* Ziel												UTF8->ASCII		BacNet Text		Textlistname									BacNet Funktion																	BacNet Textlist type												TextId		*)
		J_NC_96.IEventMessageTextsConfig.sToOffNormal	:=	fcUtfToAscii(	fcGetBcText(	GVL_BACNET.fbBacNetParameter.metGetTextListName(enTypeOfBacNetFunktionIn := enTypeOfBacNetFunktion.Type_Automationsstation,		enTypeOfBacNetTextListIn := enTypeOfBacNetTextList.EVENTMESSAGE	),	'J_NC_96_ToOffNormal'	));		
		J_NC_96.IEventMessageTextsConfig.sToFault		:=	fcUtfToAscii(	fcGetBcText(	GVL_BACNET.fbBacNetParameter.metGetTextListName(enTypeOfBacNetFunktionIn := enTypeOfBacNetFunktion.Type_Automationsstation,		enTypeOfBacNetTextListIn := enTypeOfBacNetTextList.EVENTMESSAGE	),	'J_NC_96_ToFault'		));		
		J_NC_96.IEventMessageTextsConfig.sToNormal		:=	fcUtfToAscii(	fcGetBcText(	GVL_BACNET.fbBacNetParameter.metGetTextListName(enTypeOfBacNetFunktionIn := enTypeOfBacNetFunktion.Type_Automationsstation,		enTypeOfBacNetTextListIn := enTypeOfBacNetTextList.EVENTMESSAGE	),	'J_NC_96_ToNormal'		));		
		
		(* Notification Class & Type *)
		J_NC_96.udiNotificationClass					:=  96;	
		J_NC_96.eNotifyType								:= 	WagoTypesBACnet.eBACnetNotifyType.NOTIFY_TYPE_ALARM;
		(* Ziel												Convert			BacNet Text		Textlistname									BacNet Funktion																	BacNet Textlist type												TextId		*)	
		J_NC_96.IPriority.usiToOffNormal				:= 	TO_USINT(fcUtfToAscii(	fcGetBcText(	GVL_BACNET.fbBacNetParameter.metGetTextListName(enTypeOfBacNetFunktionIn := enTypeOfBacNetFunktion.Type_Automationsstation,		enTypeOfBacNetTextListIn := enTypeOfBacNetTextList.NC	),	'J_NC_96_Prio_ToOffNormal'	)));	
		J_NC_96.IPriority.usiToFault					:= 	TO_USINT(fcUtfToAscii(	fcGetBcText(	GVL_BACNET.fbBacNetParameter.metGetTextListName(enTypeOfBacNetFunktionIn := enTypeOfBacNetFunktion.Type_Automationsstation,		enTypeOfBacNetTextListIn := enTypeOfBacNetTextList.NC	),	'J_NC_96_Prio_ToFault'		)));	
		J_NC_96.IPriority.usiToNormal					:= 	TO_USINT(fcUtfToAscii(	fcGetBcText(	GVL_BACNET.fbBacNetParameter.metGetTextListName(enTypeOfBacNetFunktionIn := enTypeOfBacNetFunktion.Type_Automationsstation,		enTypeOfBacNetTextListIn := enTypeOfBacNetTextList.NC	),	'J_NC_96_Prio_ToNormal'		)));	
		
	ELSE
		J_NC_96.Delete();
	END_IF;
	(* Get Status *)
	metCreate_J_NC_96 := J_NC_96.xIsCreated;	
END_IF;
END_METHOD

METHOD metCreate_K_NC_129 : BOOL

VAR

END_VAR
(* K_NC_129*)
IF NOT K_NC_129.xIsCreated THEN
	(* Ziel						UTF8->ASCII						OBJ_NAME_BASE			BacNet Text		Textlistname									BacNet Funktion																	BacNet Textlist type												TextId		*)
	K_NC_129._sObjectName		:=	fcUtfToAscii(Standard.CONCAT(	OBJ_NAME_BASE		,	fcGetBcText(	GVL_BACNET.fbBacNetParameter.metGetTextListName(enTypeOfBacNetFunktionIn := enTypeOfBacNetFunktion.Type_Automationsstation,		enTypeOfBacNetTextListIn := enTypeOfBacNetTextList.ENDING		),	'K_NC_129')));
	K_NC_129._sDescription	:= 	fcUtfToAscii(Standard.CONCAT(	OBJ_NAME_DESCRIPTION,	fcGetBcText(	GVL_BACNET.fbBacNetParameter.metGetTextListName(enTypeOfBacNetFunktionIn := enTypeOfBacNetFunktion.Type_Automationsstation,		enTypeOfBacNetTextListIn := enTypeOfBacNetTextList.DESCRIPTION	),	'K_NC_129')));
	(* Create Id from Base Id and Object Nr (Last nummber of Name *)	
	K_NC_129.Create(diInstance := 129);
	(* Check if Created *)
	IF K_NC_129.xIsCreated THEN
		(* Set Group *)
		K_NC_129.setPropertyGroup(WagoTypesBacNet.eBACnetPropertyIdentifier.PROP_DESCRIPTION							,WagoTypesBacNet.eBACnetPropertyUpdateGroup.GROUP_CYCLIC);
		
		(* Set Ack Req *)
		K_NC_129.IAckRequired.xToOffNormal	:= FALSE;
		K_NC_129.IAckRequired.xToFault		:= TRUE;
		K_NC_129.IAckRequired.xToNormal		:= FALSE;
		
		(* Ziel												UTF8->ASCII		BacNet Text		Textlistname									BacNet Funktion																	BacNet Textlist type												TextId		*)
		K_NC_129.IEventMessageTextsConfig.sToOffNormal	:=	fcUtfToAscii(	fcGetBcText(	GVL_BACNET.fbBacNetParameter.metGetTextListName(enTypeOfBacNetFunktionIn := enTypeOfBacNetFunktion.Type_Automationsstation,		enTypeOfBacNetTextListIn := enTypeOfBacNetTextList.EVENTMESSAGE	),	'K_NC_129_ToOffNormal'	));		
		K_NC_129.IEventMessageTextsConfig.sToFault		:=	fcUtfToAscii(	fcGetBcText(	GVL_BACNET.fbBacNetParameter.metGetTextListName(enTypeOfBacNetFunktionIn := enTypeOfBacNetFunktion.Type_Automationsstation,		enTypeOfBacNetTextListIn := enTypeOfBacNetTextList.EVENTMESSAGE	),	'K_NC_129_ToFault'		));		
		K_NC_129.IEventMessageTextsConfig.sToNormal		:=	fcUtfToAscii(	fcGetBcText(	GVL_BACNET.fbBacNetParameter.metGetTextListName(enTypeOfBacNetFunktionIn := enTypeOfBacNetFunktion.Type_Automationsstation,		enTypeOfBacNetTextListIn := enTypeOfBacNetTextList.EVENTMESSAGE	),	'K_NC_129_ToNormal'		));		
		
		(* Notification Class & Type *)
		K_NC_129.udiNotificationClass					:=  129;	
		K_NC_129.eNotifyType								:= 	WagoTypesBACnet.eBACnetNotifyType.NOTIFY_TYPE_ALARM;
		(* Ziel												Convert			BacNet Text		Textlistname									BacNet Funktion																	BacNet Textlist type												TextId		*)	
		K_NC_129.IPriority.usiToOffNormal				:= 	TO_USINT(fcUtfToAscii(	fcGetBcText(	GVL_BACNET.fbBacNetParameter.metGetTextListName(enTypeOfBacNetFunktionIn := enTypeOfBacNetFunktion.Type_Automationsstation,		enTypeOfBacNetTextListIn := enTypeOfBacNetTextList.NC	),	'K_NC_129_Prio_ToOffNormal'	)));	
		K_NC_129.IPriority.usiToFault					:= 	TO_USINT(fcUtfToAscii(	fcGetBcText(	GVL_BACNET.fbBacNetParameter.metGetTextListName(enTypeOfBacNetFunktionIn := enTypeOfBacNetFunktion.Type_Automationsstation,		enTypeOfBacNetTextListIn := enTypeOfBacNetTextList.NC	),	'K_NC_129_Prio_ToFault'		)));	
		K_NC_129.IPriority.usiToNormal					:= 	TO_USINT(fcUtfToAscii(	fcGetBcText(	GVL_BACNET.fbBacNetParameter.metGetTextListName(enTypeOfBacNetFunktionIn := enTypeOfBacNetFunktion.Type_Automationsstation,		enTypeOfBacNetTextListIn := enTypeOfBacNetTextList.NC	),	'K_NC_129_Prio_ToNormal'		)));	
		
	ELSE
		K_NC_129.Delete();
	END_IF;
	(* Get Status *)
	metCreate_K_NC_129 := K_NC_129.xIsCreated;	
END_IF;
END_METHOD

METHOD metCreate_K_NC_130 : BOOL

VAR

END_VAR
(* K_NC_130*)
IF NOT K_NC_130.xIsCreated THEN
	(* Ziel						UTF8->ASCII						OBJ_NAME_BASE			BacNet Text		Textlistname									BacNet Funktion																	BacNet Textlist type												TextId		*)
	K_NC_130._sObjectName		:=	fcUtfToAscii(Standard.CONCAT(	OBJ_NAME_BASE		,	fcGetBcText(	GVL_BACNET.fbBacNetParameter.metGetTextListName(enTypeOfBacNetFunktionIn := enTypeOfBacNetFunktion.Type_Automationsstation,		enTypeOfBacNetTextListIn := enTypeOfBacNetTextList.ENDING		),	'K_NC_130')));
	K_NC_130._sDescription	:= 	fcUtfToAscii(Standard.CONCAT(	OBJ_NAME_DESCRIPTION,	fcGetBcText(	GVL_BACNET.fbBacNetParameter.metGetTextListName(enTypeOfBacNetFunktionIn := enTypeOfBacNetFunktion.Type_Automationsstation,		enTypeOfBacNetTextListIn := enTypeOfBacNetTextList.DESCRIPTION	),	'K_NC_130')));
	(* Create Id from Base Id and Object Nr (Last nummber of Name *)	
	K_NC_130.Create(diInstance := 130);
	(* Check if Created *)
	IF K_NC_130.xIsCreated THEN
		(* Set Group *)
		K_NC_130.setPropertyGroup(WagoTypesBacNet.eBACnetPropertyIdentifier.PROP_DESCRIPTION							,WagoTypesBacNet.eBACnetPropertyUpdateGroup.GROUP_CYCLIC);
		
		(* Set Ack Req *)
		K_NC_130.IAckRequired.xToOffNormal	:= TRUE;
		K_NC_130.IAckRequired.xToFault		:= TRUE;
		K_NC_130.IAckRequired.xToNormal		:= FALSE;
		
		(* Ziel												UTF8->ASCII		BacNet Text		Textlistname									BacNet Funktion																	BacNet Textlist type												TextId		*)
		K_NC_130.IEventMessageTextsConfig.sToOffNormal	:=	fcUtfToAscii(	fcGetBcText(	GVL_BACNET.fbBacNetParameter.metGetTextListName(enTypeOfBacNetFunktionIn := enTypeOfBacNetFunktion.Type_Automationsstation,		enTypeOfBacNetTextListIn := enTypeOfBacNetTextList.EVENTMESSAGE	),	'K_NC_130_ToOffNormal'	));		
		K_NC_130.IEventMessageTextsConfig.sToFault		:=	fcUtfToAscii(	fcGetBcText(	GVL_BACNET.fbBacNetParameter.metGetTextListName(enTypeOfBacNetFunktionIn := enTypeOfBacNetFunktion.Type_Automationsstation,		enTypeOfBacNetTextListIn := enTypeOfBacNetTextList.EVENTMESSAGE	),	'K_NC_130_ToFault'		));		
		K_NC_130.IEventMessageTextsConfig.sToNormal		:=	fcUtfToAscii(	fcGetBcText(	GVL_BACNET.fbBacNetParameter.metGetTextListName(enTypeOfBacNetFunktionIn := enTypeOfBacNetFunktion.Type_Automationsstation,		enTypeOfBacNetTextListIn := enTypeOfBacNetTextList.EVENTMESSAGE	),	'K_NC_130_ToNormal'		));		
		
		(* Notification Class & Type *)
		K_NC_130.udiNotificationClass					:=  130;	
		K_NC_130.eNotifyType								:= 	WagoTypesBACnet.eBACnetNotifyType.NOTIFY_TYPE_ALARM;
		(* Ziel												Convert			BacNet Text		Textlistname									BacNet Funktion																	BacNet Textlist type												TextId		*)	
		K_NC_130.IPriority.usiToOffNormal				:= 	TO_USINT(fcUtfToAscii(	fcGetBcText(	GVL_BACNET.fbBacNetParameter.metGetTextListName(enTypeOfBacNetFunktionIn := enTypeOfBacNetFunktion.Type_Automationsstation,		enTypeOfBacNetTextListIn := enTypeOfBacNetTextList.NC	),	'K_NC_130_Prio_ToOffNormal'	)));	
		K_NC_130.IPriority.usiToFault					:= 	TO_USINT(fcUtfToAscii(	fcGetBcText(	GVL_BACNET.fbBacNetParameter.metGetTextListName(enTypeOfBacNetFunktionIn := enTypeOfBacNetFunktion.Type_Automationsstation,		enTypeOfBacNetTextListIn := enTypeOfBacNetTextList.NC	),	'K_NC_130_Prio_ToFault'		)));	
		K_NC_130.IPriority.usiToNormal					:= 	TO_USINT(fcUtfToAscii(	fcGetBcText(	GVL_BACNET.fbBacNetParameter.metGetTextListName(enTypeOfBacNetFunktionIn := enTypeOfBacNetFunktion.Type_Automationsstation,		enTypeOfBacNetTextListIn := enTypeOfBacNetTextList.NC	),	'K_NC_130_Prio_ToNormal'		)));	
		
	ELSE
		K_NC_130.Delete();
	END_IF;
	(* Get Status *)
	metCreate_K_NC_130 := K_NC_130.xIsCreated;	
END_IF;
END_METHOD

METHOD metCreate_K_NC_131 : BOOL

VAR

END_VAR
(* K_NC_131*)
IF NOT K_NC_131.xIsCreated THEN
	(* Ziel						UTF8->ASCII						OBJ_NAME_BASE			BacNet Text		Textlistname									BacNet Funktion																	BacNet Textlist type												TextId		*)
	K_NC_131._sObjectName		:=	fcUtfToAscii(Standard.CONCAT(	OBJ_NAME_BASE		,	fcGetBcText(	GVL_BACNET.fbBacNetParameter.metGetTextListName(enTypeOfBacNetFunktionIn := enTypeOfBacNetFunktion.Type_Automationsstation,		enTypeOfBacNetTextListIn := enTypeOfBacNetTextList.ENDING		),	'K_NC_131')));
	K_NC_131._sDescription	:= 	fcUtfToAscii(Standard.CONCAT(	OBJ_NAME_DESCRIPTION,	fcGetBcText(	GVL_BACNET.fbBacNetParameter.metGetTextListName(enTypeOfBacNetFunktionIn := enTypeOfBacNetFunktion.Type_Automationsstation,		enTypeOfBacNetTextListIn := enTypeOfBacNetTextList.DESCRIPTION	),	'K_NC_131')));
	(* Create Id from Base Id and Object Nr (Last nummber of Name *)	
	K_NC_131.Create(diInstance := 131);
	(* Check if Created *)
	IF K_NC_131.xIsCreated THEN
		(* Set Group *)
		K_NC_131.setPropertyGroup(WagoTypesBacNet.eBACnetPropertyIdentifier.PROP_DESCRIPTION							,WagoTypesBacNet.eBACnetPropertyUpdateGroup.GROUP_CYCLIC);
		
		(* Set Ack Req *)
		K_NC_131.IAckRequired.xToOffNormal	:= TRUE;
		K_NC_131.IAckRequired.xToFault		:= TRUE;
		K_NC_131.IAckRequired.xToNormal		:= TRUE;
		
		(* Ziel												UTF8->ASCII		BacNet Text		Textlistname									BacNet Funktion																	BacNet Textlist type												TextId		*)
		K_NC_131.IEventMessageTextsConfig.sToOffNormal	:=	fcUtfToAscii(	fcGetBcText(	GVL_BACNET.fbBacNetParameter.metGetTextListName(enTypeOfBacNetFunktionIn := enTypeOfBacNetFunktion.Type_Automationsstation,		enTypeOfBacNetTextListIn := enTypeOfBacNetTextList.EVENTMESSAGE	),	'K_NC_131_ToOffNormal'	));		
		K_NC_131.IEventMessageTextsConfig.sToFault		:=	fcUtfToAscii(	fcGetBcText(	GVL_BACNET.fbBacNetParameter.metGetTextListName(enTypeOfBacNetFunktionIn := enTypeOfBacNetFunktion.Type_Automationsstation,		enTypeOfBacNetTextListIn := enTypeOfBacNetTextList.EVENTMESSAGE	),	'K_NC_131_ToFault'		));		
		K_NC_131.IEventMessageTextsConfig.sToNormal		:=	fcUtfToAscii(	fcGetBcText(	GVL_BACNET.fbBacNetParameter.metGetTextListName(enTypeOfBacNetFunktionIn := enTypeOfBacNetFunktion.Type_Automationsstation,		enTypeOfBacNetTextListIn := enTypeOfBacNetTextList.EVENTMESSAGE	),	'K_NC_131_ToNormal'		));		
		
		(* Notification Class & Type *)
		K_NC_131.udiNotificationClass					:=  131;	
		K_NC_131.eNotifyType							:= 	WagoTypesBACnet.eBACnetNotifyType.NOTIFY_TYPE_ALARM;
		(* Ziel												Convert			BacNet Text		Textlistname									BacNet Funktion																	BacNet Textlist type												TextId		*)	
		K_NC_131.IPriority.usiToOffNormal				:= 	TO_USINT(fcUtfToAscii(	fcGetBcText(	GVL_BACNET.fbBacNetParameter.metGetTextListName(enTypeOfBacNetFunktionIn := enTypeOfBacNetFunktion.Type_Automationsstation,		enTypeOfBacNetTextListIn := enTypeOfBacNetTextList.NC	),	'K_NC_131_Prio_ToOffNormal'	)));	
		K_NC_131.IPriority.usiToFault					:= 	TO_USINT(fcUtfToAscii(	fcGetBcText(	GVL_BACNET.fbBacNetParameter.metGetTextListName(enTypeOfBacNetFunktionIn := enTypeOfBacNetFunktion.Type_Automationsstation,		enTypeOfBacNetTextListIn := enTypeOfBacNetTextList.NC	),	'K_NC_131_Prio_ToFault'		)));	
		K_NC_131.IPriority.usiToNormal					:= 	TO_USINT(fcUtfToAscii(	fcGetBcText(	GVL_BACNET.fbBacNetParameter.metGetTextListName(enTypeOfBacNetFunktionIn := enTypeOfBacNetFunktion.Type_Automationsstation,		enTypeOfBacNetTextListIn := enTypeOfBacNetTextList.NC	),	'K_NC_131_Prio_ToNormal'		)));	
		
	ELSE
		K_NC_131.Delete();
	END_IF;
	(* Get Status *)
	metCreate_K_NC_131 := K_NC_131.xIsCreated;	
END_IF;
END_METHOD

METHOD metCreate_A_DV_1 : BOOL

VAR

END_VAR
(* A_DV_1*)
IF NOT A_DV_1.xIsCreated THEN
	(* Ziel						UTF8->ASCII						OBJ_NAME_BASE			BacNet Text		Textlistname									BacNet Funktion																	BacNet Textlist type												TextId		*)
	A_DV_1._sObjectName		:=	fcUtfToAscii(Standard.CONCAT(	OBJ_NAME_BASE		,	fcGetBcText(	GVL_BACNET.fbBacNetParameter.metGetTextListName(enTypeOfBacNetFunktionIn := enTypeOfBacNetFunktion.Type_Automationsstation,		enTypeOfBacNetTextListIn := enTypeOfBacNetTextList.ENDING		),	'A_DV_1')));
	A_DV_1._sDescription	:= 	fcUtfToAscii(Standard.CONCAT(	OBJ_NAME_DESCRIPTION,	fcGetBcText(	GVL_BACNET.fbBacNetParameter.metGetTextListName(enTypeOfBacNetFunktionIn := enTypeOfBacNetFunktion.Type_Automationsstation,		enTypeOfBacNetTextListIn := enTypeOfBacNetTextList.DESCRIPTION	),	'A_DV_1')));
	(* Create Id from Base Id and Object Nr (Last nummber of Name *)	
	A_DV_1.Create(diInstance := GVL_BACNET.fbBacNetParameter.fbdiDeviceId.proValue);
	(* Check if Created *)
	IF A_DV_1.xIsCreated THEN
		(* XML Override *)
		fcXMLDeviceOverride(A_DV_1,GVL_BACNET.fbBacNetParameter.fbdiDeviceId.proValue,A_DV_1._sObjectName);
		(* Set Group *)
		A_DV_1.setPropertyGroup(WagoTypesBacNet.eBACnetPropertyIdentifier.PROP_PRESENT_VALUE						,WagoTypesBacNet.eBACnetPropertyUpdateGroup.GROUP_CYCLIC);
		A_DV_1.setPropertyGroup(WagoTypesBacNet.eBACnetPropertyIdentifier.PROP_PRIORITY_ARRAY						,WagoTypesBacNet.eBACnetPropertyUpdateGroup.GROUP_CYCLIC);
		A_DV_1.setPropertyGroup(WagoTypesBacNet.eBACnetPropertyIdentifier.PROP_ELAPSED_ACTIVE_TIME					,WagoTypesBacNet.eBACnetPropertyUpdateGroup.GROUP_CYCLIC);
		A_DV_1.setPropertyGroup(WagoTypesBacNet.eBACnetPropertyIdentifier.PROP_DESCRIPTION							,WagoTypesBacNet.eBACnetPropertyUpdateGroup.GROUP_CYCLIC);
		A_DV_1.setPropertyGroup(WagoTypesBacNet.eBACnetPropertyIdentifier.PROP_EVENT_MESSAGE_TEXTS_CONFIG			,WagoTypesBacNet.eBACnetPropertyUpdateGroup.GROUP_CYCLIC);
		
	ELSE
		A_DV_1.Delete();
	END_IF;
	(* Get Status *)
	metCreate_A_DV_1 := A_DV_1.xIsCreated;	
END_IF;
END_METHOD

METHOD metCreate_B_CL_1 : BOOL

VAR

END_VAR
(* B_CL_1*)
IF NOT B_CL_1.xIsCreated THEN
	(* Ziel						UTF8->ASCII						OBJ_NAME_BASE			BacNet Text		Textlistname									BacNet Funktion																	BacNet Textlist type												TextId		*)
	B_CL_1._sObjectName		:=	fcUtfToAscii(Standard.CONCAT(	OBJ_NAME_BASE		,	fcGetBcText(	GVL_BACNET.fbBacNetParameter.metGetTextListName(enTypeOfBacNetFunktionIn := enTypeOfBacNetFunktion.Type_Automationsstation,		enTypeOfBacNetTextListIn := enTypeOfBacNetTextList.ENDING		),	'B_CL_1')));
	B_CL_1._sDescription	:= 	fcUtfToAscii(Standard.CONCAT(	OBJ_NAME_DESCRIPTION,	fcGetBcText(	GVL_BACNET.fbBacNetParameter.metGetTextListName(enTypeOfBacNetFunktionIn := enTypeOfBacNetFunktion.Type_Automationsstation,		enTypeOfBacNetTextListIn := enTypeOfBacNetTextList.DESCRIPTION	),	'B_CL_1')));
	(* Create Id from Base Id and Object Nr (Last nummber of Name *)	
	B_CL_1.Create(diInstance := TO_DINT(Standard.CONCAT(TO_STRING(dwOBJ_ID_BASE),'1')));
	(* Check if Created *)
	IF B_CL_1.xIsCreated THEN
		(* Set Group *)
		B_CL_1.setPropertyGroup(WagoTypesBacNet.eBACnetPropertyIdentifier.PROP_DESCRIPTION							,WagoTypesBacNet.eBACnetPropertyUpdateGroup.GROUP_CYCLIC);
		
	ELSE
		B_CL_1.Delete();
	END_IF;
	(* Get Status *)
	metCreate_B_CL_1 := B_CL_1.xIsCreated;	
END_IF;
END_METHOD

METHOD metCreate_C_CL_2 : BOOL

VAR

END_VAR
(* C_CL_2*)
IF NOT C_CL_2.xIsCreated THEN
	(* Ziel						UTF8->ASCII						OBJ_NAME_BASE			BacNet Text		Textlistname									BacNet Funktion																	BacNet Textlist type												TextId		*)
	C_CL_2._sObjectName		:=	fcUtfToAscii(Standard.CONCAT(	OBJ_NAME_BASE		,	fcGetBcText(	GVL_BACNET.fbBacNetParameter.metGetTextListName(enTypeOfBacNetFunktionIn := enTypeOfBacNetFunktion.Type_Automationsstation,		enTypeOfBacNetTextListIn := enTypeOfBacNetTextList.ENDING		),	'C_CL_2')));
	C_CL_2._sDescription	:= 	fcUtfToAscii(Standard.CONCAT(	OBJ_NAME_DESCRIPTION,	fcGetBcText(	GVL_BACNET.fbBacNetParameter.metGetTextListName(enTypeOfBacNetFunktionIn := enTypeOfBacNetFunktion.Type_Automationsstation,		enTypeOfBacNetTextListIn := enTypeOfBacNetTextList.DESCRIPTION	),	'C_CL_2')));
	(* Create Id from Base Id and Object Nr (Last nummber of Name *)	
	C_CL_2.Create(diInstance := TO_DINT(Standard.CONCAT(TO_STRING(dwOBJ_ID_BASE),'2')));
	(* Check if Created *)
	IF C_CL_2.xIsCreated THEN
		(* Set Group *)
		C_CL_2.setPropertyGroup(WagoTypesBacNet.eBACnetPropertyIdentifier.PROP_DESCRIPTION							,WagoTypesBacNet.eBACnetPropertyUpdateGroup.GROUP_CYCLIC);
		
	ELSE
		C_CL_2.Delete();
	END_IF;
	(* Get Status *)
	metCreate_C_CL_2 := C_CL_2.xIsCreated;	
END_IF;
END_METHOD

METHOD metCreate_D_CL_3 : BOOL

VAR

END_VAR
(* D_CL_3*)
IF NOT D_CL_3.xIsCreated THEN
	(* Ziel						UTF8->ASCII						OBJ_NAME_BASE			BacNet Text		Textlistname									BacNet Funktion																	BacNet Textlist type												TextId		*)
	D_CL_3._sObjectName		:=	fcUtfToAscii(Standard.CONCAT(	OBJ_NAME_BASE		,	fcGetBcText(	GVL_BACNET.fbBacNetParameter.metGetTextListName(enTypeOfBacNetFunktionIn := enTypeOfBacNetFunktion.Type_Automationsstation,		enTypeOfBacNetTextListIn := enTypeOfBacNetTextList.ENDING		),	'D_CL_3')));
	D_CL_3._sDescription	:= 	fcUtfToAscii(Standard.CONCAT(	OBJ_NAME_DESCRIPTION,	fcGetBcText(	GVL_BACNET.fbBacNetParameter.metGetTextListName(enTypeOfBacNetFunktionIn := enTypeOfBacNetFunktion.Type_Automationsstation,		enTypeOfBacNetTextListIn := enTypeOfBacNetTextList.DESCRIPTION	),	'D_CL_3')));
	(* Create Id from Base Id and Object Nr (Last nummber of Name *)	
	D_CL_3.Create(diInstance := TO_DINT(Standard.CONCAT(TO_STRING(dwOBJ_ID_BASE),'3')));
	(* Check if Created *)
	IF D_CL_3.xIsCreated THEN
		(* Set Group *)
		D_CL_3.setPropertyGroup(WagoTypesBacNet.eBACnetPropertyIdentifier.PROP_DESCRIPTION							,WagoTypesBacNet.eBACnetPropertyUpdateGroup.GROUP_CYCLIC);
		
	ELSE
		D_CL_3.Delete();
	END_IF;
	(* Get Status *)
	metCreate_D_CL_3 := D_CL_3.xIsCreated;	
END_IF;
END_METHOD

METHOD metCreate_E_CL_4 : BOOL

VAR

END_VAR
(* E_CL_4*)
IF NOT E_CL_4.xIsCreated THEN
	(* Ziel						UTF8->ASCII						OBJ_NAME_BASE			BacNet Text		Textlistname									BacNet Funktion																	BacNet Textlist type												TextId		*)
	E_CL_4._sObjectName		:=	fcUtfToAscii(Standard.CONCAT(	OBJ_NAME_BASE		,	fcGetBcText(	GVL_BACNET.fbBacNetParameter.metGetTextListName(enTypeOfBacNetFunktionIn := enTypeOfBacNetFunktion.Type_Automationsstation,		enTypeOfBacNetTextListIn := enTypeOfBacNetTextList.ENDING		),	'E_CL_4')));
	E_CL_4._sDescription	:= 	fcUtfToAscii(Standard.CONCAT(	OBJ_NAME_DESCRIPTION,	fcGetBcText(	GVL_BACNET.fbBacNetParameter.metGetTextListName(enTypeOfBacNetFunktionIn := enTypeOfBacNetFunktion.Type_Automationsstation,		enTypeOfBacNetTextListIn := enTypeOfBacNetTextList.DESCRIPTION	),	'E_CL_4')));
	(* Create Id from Base Id and Object Nr (Last nummber of Name *)	
	E_CL_4.Create(diInstance := TO_DINT(Standard.CONCAT(TO_STRING(dwOBJ_ID_BASE),'4')));
	(* Check if Created *)
	IF E_CL_4.xIsCreated THEN
		(* Set Group *)
		E_CL_4.setPropertyGroup(WagoTypesBacNet.eBACnetPropertyIdentifier.PROP_DESCRIPTION							,WagoTypesBacNet.eBACnetPropertyUpdateGroup.GROUP_CYCLIC);
		
	ELSE
		E_CL_4.Delete();
	END_IF;
	(* Get Status *)
	metCreate_E_CL_4 := E_CL_4.xIsCreated;	
END_IF;
END_METHOD

METHOD metCreate_F_EL_1 : BOOL

VAR

END_VAR
(* F_EL_1*)
IF NOT F_EL_1.xIsCreated THEN
	(* Ziel						UTF8->ASCII						OBJ_NAME_BASE			BacNet Text		Textlistname									BacNet Funktion																	BacNet Textlist type												TextId		*)
	F_EL_1._sObjectName		:=	fcUtfToAscii(Standard.CONCAT(	OBJ_NAME_BASE		,	fcGetBcText(	GVL_BACNET.fbBacNetParameter.metGetTextListName(enTypeOfBacNetFunktionIn := enTypeOfBacNetFunktion.Type_Automationsstation,		enTypeOfBacNetTextListIn := enTypeOfBacNetTextList.ENDING		),	'F_EL_1')));
	F_EL_1._sDescription	:= 	fcUtfToAscii(Standard.CONCAT(	OBJ_NAME_DESCRIPTION,	fcGetBcText(	GVL_BACNET.fbBacNetParameter.metGetTextListName(enTypeOfBacNetFunktionIn := enTypeOfBacNetFunktion.Type_Automationsstation,		enTypeOfBacNetTextListIn := enTypeOfBacNetTextList.DESCRIPTION	),	'F_EL_1')));
	(* Create Id from Base Id and Object Nr (Last nummber of Name *)	
	F_EL_1.Create(diInstance := TO_DINT(Standard.CONCAT(TO_STRING(dwOBJ_ID_BASE),'1')));
	(* Check if Created *)
	IF F_EL_1.xIsCreated THEN
		(* Set Group *)
		F_EL_1.setPropertyGroup(WagoTypesBacNet.eBACnetPropertyIdentifier.PROP_DESCRIPTION							,WagoTypesBacNet.eBACnetPropertyUpdateGroup.GROUP_CYCLIC);
		
	ELSE
		F_EL_1.Delete();
	END_IF;
	(* Get Status *)
	metCreate_F_EL_1 := F_EL_1.xIsCreated;	
END_IF;
END_METHOD

METHOD metCreate_G_NC_1 : BOOL

VAR

END_VAR
(* G_NC_1*)
IF NOT G_NC_1.xIsCreated THEN
	(* Ziel						UTF8->ASCII						OBJ_NAME_BASE			BacNet Text		Textlistname									BacNet Funktion																	BacNet Textlist type												TextId		*)
	G_NC_1._sObjectName		:=	fcUtfToAscii(Standard.CONCAT(	OBJ_NAME_BASE		,	fcGetBcText(	GVL_BACNET.fbBacNetParameter.metGetTextListName(enTypeOfBacNetFunktionIn := enTypeOfBacNetFunktion.Type_Automationsstation,		enTypeOfBacNetTextListIn := enTypeOfBacNetTextList.ENDING		),	'G_NC_1')));
	G_NC_1._sDescription	:= 	fcUtfToAscii(Standard.CONCAT(	OBJ_NAME_DESCRIPTION,	fcGetBcText(	GVL_BACNET.fbBacNetParameter.metGetTextListName(enTypeOfBacNetFunktionIn := enTypeOfBacNetFunktion.Type_Automationsstation,		enTypeOfBacNetTextListIn := enTypeOfBacNetTextList.DESCRIPTION	),	'G_NC_1')));
	(* Create Id from Base Id and Object Nr (Last nummber of Name *)	
	G_NC_1.Create(diInstance := 1);
	(* Check if Created *)
	IF G_NC_1.xIsCreated THEN
		(* Set Group *)
		G_NC_1.setPropertyGroup(WagoTypesBacNet.eBACnetPropertyIdentifier.PROP_DESCRIPTION							,WagoTypesBacNet.eBACnetPropertyUpdateGroup.GROUP_CYCLIC);
		
		(* Set Ack Req *)
		G_NC_1.IAckRequired.xToOffNormal	:= FALSE;
		G_NC_1.IAckRequired.xToFault		:= FALSE;
		G_NC_1.IAckRequired.xToNormal		:= FALSE;
		
		(* Ziel												UTF8->ASCII		BacNet Text		Textlistname									BacNet Funktion																	BacNet Textlist type												TextId		*)
		G_NC_1.IEventMessageTextsConfig.sToOffNormal	:=	fcUtfToAscii(	fcGetBcText(	GVL_BACNET.fbBacNetParameter.metGetTextListName(enTypeOfBacNetFunktionIn := enTypeOfBacNetFunktion.Type_Automationsstation,		enTypeOfBacNetTextListIn := enTypeOfBacNetTextList.EVENTMESSAGE	),	'G_NC_1_ToOffNormal'	));		
		G_NC_1.IEventMessageTextsConfig.sToFault		:=	fcUtfToAscii(	fcGetBcText(	GVL_BACNET.fbBacNetParameter.metGetTextListName(enTypeOfBacNetFunktionIn := enTypeOfBacNetFunktion.Type_Automationsstation,		enTypeOfBacNetTextListIn := enTypeOfBacNetTextList.EVENTMESSAGE	),	'G_NC_1_ToFault'		));		
		G_NC_1.IEventMessageTextsConfig.sToNormal		:=	fcUtfToAscii(	fcGetBcText(	GVL_BACNET.fbBacNetParameter.metGetTextListName(enTypeOfBacNetFunktionIn := enTypeOfBacNetFunktion.Type_Automationsstation,		enTypeOfBacNetTextListIn := enTypeOfBacNetTextList.EVENTMESSAGE	),	'G_NC_1_ToNormal'		));		
		
		(* Notification Class & Type *)
		G_NC_1.udiNotificationClass						:= 	1;	
		G_NC_1.eNotifyType								:= 	WagoTypesBACnet.eBACnetNotifyType.NOTIFY_TYPE_ALARM;
		(* Ziel												Convert			BacNet Text		Textlistname									BacNet Funktion																	BacNet Textlist type												TextId		*)	
		G_NC_1.IPriority.usiToOffNormal					:= 	TO_USINT(fcUtfToAscii(	fcGetBcText(	GVL_BACNET.fbBacNetParameter.metGetTextListName(enTypeOfBacNetFunktionIn := enTypeOfBacNetFunktion.Type_Automationsstation,		enTypeOfBacNetTextListIn := enTypeOfBacNetTextList.NC	),	'G_NC_1_Prio_ToOffNormal'	)));	
		G_NC_1.IPriority.usiToFault						:= 	TO_USINT(fcUtfToAscii(	fcGetBcText(	GVL_BACNET.fbBacNetParameter.metGetTextListName(enTypeOfBacNetFunktionIn := enTypeOfBacNetFunktion.Type_Automationsstation,		enTypeOfBacNetTextListIn := enTypeOfBacNetTextList.NC	),	'G_NC_1_Prio_ToFault'		)));	
		G_NC_1.IPriority.usiToNormal					:= 	TO_USINT(fcUtfToAscii(	fcGetBcText(	GVL_BACNET.fbBacNetParameter.metGetTextListName(enTypeOfBacNetFunktionIn := enTypeOfBacNetFunktion.Type_Automationsstation,		enTypeOfBacNetTextListIn := enTypeOfBacNetTextList.NC	),	'G_NC_1_Prio_ToNormal'		)));	
		
	ELSE
		G_NC_1.Delete();
	END_IF;
	(* Get Status *)
	metCreate_G_NC_1 := G_NC_1.xIsCreated;	
END_IF;
END_METHOD

METHOD metCreate_G_NC_2 : BOOL

VAR

END_VAR
(* G_NC_2*)
IF NOT G_NC_2.xIsCreated THEN
	(* Ziel						UTF8->ASCII						OBJ_NAME_BASE			BacNet Text		Textlistname									BacNet Funktion																	BacNet Textlist type												TextId		*)
	G_NC_2._sObjectName		:=	fcUtfToAscii(Standard.CONCAT(	OBJ_NAME_BASE		,	fcGetBcText(	GVL_BACNET.fbBacNetParameter.metGetTextListName(enTypeOfBacNetFunktionIn := enTypeOfBacNetFunktion.Type_Automationsstation,		enTypeOfBacNetTextListIn := enTypeOfBacNetTextList.ENDING		),	'G_NC_2')));
	G_NC_2._sDescription	:= 	fcUtfToAscii(Standard.CONCAT(	OBJ_NAME_DESCRIPTION,	fcGetBcText(	GVL_BACNET.fbBacNetParameter.metGetTextListName(enTypeOfBacNetFunktionIn := enTypeOfBacNetFunktion.Type_Automationsstation,		enTypeOfBacNetTextListIn := enTypeOfBacNetTextList.DESCRIPTION	),	'G_NC_2')));
	(* Create Id from Base Id and Object Nr (Last nummber of Name *)	
	G_NC_2.Create(diInstance := 2);
	(* Check if Created *)
	IF G_NC_2.xIsCreated THEN
		(* Set Group *)
		G_NC_2.setPropertyGroup(WagoTypesBacNet.eBACnetPropertyIdentifier.PROP_DESCRIPTION							,WagoTypesBacNet.eBACnetPropertyUpdateGroup.GROUP_CYCLIC);
		
		(* Set Ack Req *)
		G_NC_2.IAckRequired.xToOffNormal	:= FALSE;
		G_NC_2.IAckRequired.xToFault		:= TRUE;
		G_NC_2.IAckRequired.xToNormal		:= FALSE;
		
		(* Ziel												UTF8->ASCII		BacNet Text		Textlistname									BacNet Funktion																	BacNet Textlist type												TextId		*)
		G_NC_2.IEventMessageTextsConfig.sToOffNormal	:=	fcUtfToAscii(	fcGetBcText(	GVL_BACNET.fbBacNetParameter.metGetTextListName(enTypeOfBacNetFunktionIn := enTypeOfBacNetFunktion.Type_Automationsstation,		enTypeOfBacNetTextListIn := enTypeOfBacNetTextList.EVENTMESSAGE	),	'G_NC_2_ToOffNormal'	));		
		G_NC_2.IEventMessageTextsConfig.sToFault		:=	fcUtfToAscii(	fcGetBcText(	GVL_BACNET.fbBacNetParameter.metGetTextListName(enTypeOfBacNetFunktionIn := enTypeOfBacNetFunktion.Type_Automationsstation,		enTypeOfBacNetTextListIn := enTypeOfBacNetTextList.EVENTMESSAGE	),	'G_NC_2_ToFault'		));		
		G_NC_2.IEventMessageTextsConfig.sToNormal		:=	fcUtfToAscii(	fcGetBcText(	GVL_BACNET.fbBacNetParameter.metGetTextListName(enTypeOfBacNetFunktionIn := enTypeOfBacNetFunktion.Type_Automationsstation,		enTypeOfBacNetTextListIn := enTypeOfBacNetTextList.EVENTMESSAGE	),	'G_NC_2_ToNormal'		));		
		
		(* Notification Class & Type *)
		G_NC_2.udiNotificationClass						:= 	2;	
		G_NC_2.eNotifyType								:= 	WagoTypesBACnet.eBACnetNotifyType.NOTIFY_TYPE_ALARM;
		(* Ziel												Convert			BacNet Text		Textlistname									BacNet Funktion																	BacNet Textlist type												TextId		*)	
		G_NC_2.IPriority.usiToOffNormal					:= 	TO_USINT(fcUtfToAscii(	fcGetBcText(	GVL_BACNET.fbBacNetParameter.metGetTextListName(enTypeOfBacNetFunktionIn := enTypeOfBacNetFunktion.Type_Automationsstation,		enTypeOfBacNetTextListIn := enTypeOfBacNetTextList.NC	),	'G_NC_2_Prio_ToOffNormal'	)));	
		G_NC_2.IPriority.usiToFault						:= 	TO_USINT(fcUtfToAscii(	fcGetBcText(	GVL_BACNET.fbBacNetParameter.metGetTextListName(enTypeOfBacNetFunktionIn := enTypeOfBacNetFunktion.Type_Automationsstation,		enTypeOfBacNetTextListIn := enTypeOfBacNetTextList.NC	),	'G_NC_2_Prio_ToFault'		)));	
		G_NC_2.IPriority.usiToNormal					:= 	TO_USINT(fcUtfToAscii(	fcGetBcText(	GVL_BACNET.fbBacNetParameter.metGetTextListName(enTypeOfBacNetFunktionIn := enTypeOfBacNetFunktion.Type_Automationsstation,		enTypeOfBacNetTextListIn := enTypeOfBacNetTextList.NC	),	'G_NC_2_Prio_ToNormal'		)));	
		
	ELSE
		G_NC_2.Delete();
	END_IF;
	(* Get Status *)
	metCreate_G_NC_2 := G_NC_2.xIsCreated;	
END_IF;
END_METHOD

METHOD metCreate_G_NC_3 : BOOL

VAR

END_VAR
(* G_NC_3*)
IF NOT G_NC_3.xIsCreated THEN
	(* Ziel						UTF8->ASCII						OBJ_NAME_BASE			BacNet Text		Textlistname									BacNet Funktion																	BacNet Textlist type												TextId		*)
	G_NC_3._sObjectName		:=	fcUtfToAscii(Standard.CONCAT(	OBJ_NAME_BASE		,	fcGetBcText(	GVL_BACNET.fbBacNetParameter.metGetTextListName(enTypeOfBacNetFunktionIn := enTypeOfBacNetFunktion.Type_Automationsstation,		enTypeOfBacNetTextListIn := enTypeOfBacNetTextList.ENDING		),	'G_NC_3')));
	G_NC_3._sDescription	:= 	fcUtfToAscii(Standard.CONCAT(	OBJ_NAME_DESCRIPTION,	fcGetBcText(	GVL_BACNET.fbBacNetParameter.metGetTextListName(enTypeOfBacNetFunktionIn := enTypeOfBacNetFunktion.Type_Automationsstation,		enTypeOfBacNetTextListIn := enTypeOfBacNetTextList.DESCRIPTION	),	'G_NC_3')));
	(* Create Id from Base Id and Object Nr (Last nummber of Name *)	
	G_NC_3.Create(diInstance := 3);
	(* Check if Created *)
	IF G_NC_3.xIsCreated THEN
		(* Set Group *)
		G_NC_3.setPropertyGroup(WagoTypesBacNet.eBACnetPropertyIdentifier.PROP_DESCRIPTION							,WagoTypesBacNet.eBACnetPropertyUpdateGroup.GROUP_CYCLIC);
		
		(* Set Ack Req *)
		G_NC_3.IAckRequired.xToOffNormal	:= TRUE;
		G_NC_3.IAckRequired.xToFault		:= TRUE;
		G_NC_3.IAckRequired.xToNormal		:= FALSE;
		
		(* Ziel												UTF8->ASCII		BacNet Text		Textlistname									BacNet Funktion																	BacNet Textlist type												TextId		*)
		G_NC_3.IEventMessageTextsConfig.sToOffNormal	:=	fcUtfToAscii(	fcGetBcText(	GVL_BACNET.fbBacNetParameter.metGetTextListName(enTypeOfBacNetFunktionIn := enTypeOfBacNetFunktion.Type_Automationsstation,		enTypeOfBacNetTextListIn := enTypeOfBacNetTextList.EVENTMESSAGE	),	'G_NC_3_ToOffNormal'	));		
		G_NC_3.IEventMessageTextsConfig.sToFault		:=	fcUtfToAscii(	fcGetBcText(	GVL_BACNET.fbBacNetParameter.metGetTextListName(enTypeOfBacNetFunktionIn := enTypeOfBacNetFunktion.Type_Automationsstation,		enTypeOfBacNetTextListIn := enTypeOfBacNetTextList.EVENTMESSAGE	),	'G_NC_3_ToFault'		));		
		G_NC_3.IEventMessageTextsConfig.sToNormal		:=	fcUtfToAscii(	fcGetBcText(	GVL_BACNET.fbBacNetParameter.metGetTextListName(enTypeOfBacNetFunktionIn := enTypeOfBacNetFunktion.Type_Automationsstation,		enTypeOfBacNetTextListIn := enTypeOfBacNetTextList.EVENTMESSAGE	),	'G_NC_3_ToNormal'		));		
		
		(* Notification Class & Type *)
		G_NC_3.udiNotificationClass						:= 	3;	
		G_NC_3.eNotifyType								:= 	WagoTypesBACnet.eBACnetNotifyType.NOTIFY_TYPE_ALARM;
		(* Ziel												Convert			BacNet Text		Textlistname									BacNet Funktion																	BacNet Textlist type												TextId		*)	
		G_NC_3.IPriority.usiToOffNormal					:= 	TO_USINT(fcUtfToAscii(	fcGetBcText(	GVL_BACNET.fbBacNetParameter.metGetTextListName(enTypeOfBacNetFunktionIn := enTypeOfBacNetFunktion.Type_Automationsstation,		enTypeOfBacNetTextListIn := enTypeOfBacNetTextList.NC	),	'G_NC_3_Prio_ToOffNormal'	)));	
		G_NC_3.IPriority.usiToFault						:= 	TO_USINT(fcUtfToAscii(	fcGetBcText(	GVL_BACNET.fbBacNetParameter.metGetTextListName(enTypeOfBacNetFunktionIn := enTypeOfBacNetFunktion.Type_Automationsstation,		enTypeOfBacNetTextListIn := enTypeOfBacNetTextList.NC	),	'G_NC_3_Prio_ToFault'		)));	
		G_NC_3.IPriority.usiToNormal					:= 	TO_USINT(fcUtfToAscii(	fcGetBcText(	GVL_BACNET.fbBacNetParameter.metGetTextListName(enTypeOfBacNetFunktionIn := enTypeOfBacNetFunktion.Type_Automationsstation,		enTypeOfBacNetTextListIn := enTypeOfBacNetTextList.NC	),	'G_NC_3_Prio_ToNormal'		)));	
		
	ELSE
		G_NC_3.Delete();
	END_IF;
	(* Get Status *)
	metCreate_G_NC_3 := G_NC_3.xIsCreated;	
END_IF;
END_METHOD

METHOD metCreate_G_NC_4 : BOOL

VAR

END_VAR
(* G_NC_4*)
IF NOT G_NC_4.xIsCreated THEN
	(* Ziel						UTF8->ASCII						OBJ_NAME_BASE			BacNet Text		Textlistname									BacNet Funktion																	BacNet Textlist type												TextId		*)
	G_NC_4._sObjectName		:=	fcUtfToAscii(Standard.CONCAT(	OBJ_NAME_BASE		,	fcGetBcText(	GVL_BACNET.fbBacNetParameter.metGetTextListName(enTypeOfBacNetFunktionIn := enTypeOfBacNetFunktion.Type_Automationsstation,		enTypeOfBacNetTextListIn := enTypeOfBacNetTextList.ENDING		),	'G_NC_4')));
	G_NC_4._sDescription	:= 	fcUtfToAscii(Standard.CONCAT(	OBJ_NAME_DESCRIPTION,	fcGetBcText(	GVL_BACNET.fbBacNetParameter.metGetTextListName(enTypeOfBacNetFunktionIn := enTypeOfBacNetFunktion.Type_Automationsstation,		enTypeOfBacNetTextListIn := enTypeOfBacNetTextList.DESCRIPTION	),	'G_NC_4')));
	(* Create Id from Base Id and Object Nr (Last nummber of Name *)	
	G_NC_4.Create(diInstance := 4);
	(* Check if Created *)
	IF G_NC_4.xIsCreated THEN
		(* Set Group *)
		G_NC_4.setPropertyGroup(WagoTypesBacNet.eBACnetPropertyIdentifier.PROP_DESCRIPTION							,WagoTypesBacNet.eBACnetPropertyUpdateGroup.GROUP_CYCLIC);
		
		(* Set Ack Req *)
		G_NC_4.IAckRequired.xToOffNormal	:= TRUE;
		G_NC_4.IAckRequired.xToFault		:= TRUE;
		G_NC_4.IAckRequired.xToNormal		:= TRUE;
		
		(* Ziel												UTF8->ASCII		BacNet Text		Textlistname									BacNet Funktion																	BacNet Textlist type												TextId		*)
		G_NC_4.IEventMessageTextsConfig.sToOffNormal	:=	fcUtfToAscii(	fcGetBcText(	GVL_BACNET.fbBacNetParameter.metGetTextListName(enTypeOfBacNetFunktionIn := enTypeOfBacNetFunktion.Type_Automationsstation,		enTypeOfBacNetTextListIn := enTypeOfBacNetTextList.EVENTMESSAGE	),	'G_NC_4_ToOffNormal'	));		
		G_NC_4.IEventMessageTextsConfig.sToFault		:=	fcUtfToAscii(	fcGetBcText(	GVL_BACNET.fbBacNetParameter.metGetTextListName(enTypeOfBacNetFunktionIn := enTypeOfBacNetFunktion.Type_Automationsstation,		enTypeOfBacNetTextListIn := enTypeOfBacNetTextList.EVENTMESSAGE	),	'G_NC_4_ToFault'		));		
		G_NC_4.IEventMessageTextsConfig.sToNormal		:=	fcUtfToAscii(	fcGetBcText(	GVL_BACNET.fbBacNetParameter.metGetTextListName(enTypeOfBacNetFunktionIn := enTypeOfBacNetFunktion.Type_Automationsstation,		enTypeOfBacNetTextListIn := enTypeOfBacNetTextList.EVENTMESSAGE	),	'G_NC_4_ToNormal'		));		
		
		(* Notification Class & Type *)
		G_NC_4.udiNotificationClass						:= 	4;	
		G_NC_4.eNotifyType								:= 	WagoTypesBACnet.eBACnetNotifyType.NOTIFY_TYPE_ALARM;
		(* Ziel												Convert			BacNet Text		Textlistname									BacNet Funktion																	BacNet Textlist type												TextId		*)	
		G_NC_4.IPriority.usiToOffNormal					:= 	TO_USINT(fcUtfToAscii(	fcGetBcText(	GVL_BACNET.fbBacNetParameter.metGetTextListName(enTypeOfBacNetFunktionIn := enTypeOfBacNetFunktion.Type_Automationsstation,		enTypeOfBacNetTextListIn := enTypeOfBacNetTextList.NC	),	'G_NC_4_Prio_ToOffNormal'	)));	
		G_NC_4.IPriority.usiToFault						:= 	TO_USINT(fcUtfToAscii(	fcGetBcText(	GVL_BACNET.fbBacNetParameter.metGetTextListName(enTypeOfBacNetFunktionIn := enTypeOfBacNetFunktion.Type_Automationsstation,		enTypeOfBacNetTextListIn := enTypeOfBacNetTextList.NC	),	'G_NC_4_Prio_ToFault'		)));	
		G_NC_4.IPriority.usiToNormal					:= 	TO_USINT(fcUtfToAscii(	fcGetBcText(	GVL_BACNET.fbBacNetParameter.metGetTextListName(enTypeOfBacNetFunktionIn := enTypeOfBacNetFunktion.Type_Automationsstation,		enTypeOfBacNetTextListIn := enTypeOfBacNetTextList.NC	),	'G_NC_4_Prio_ToNormal'		)));	
		
	ELSE
		G_NC_4.Delete();
	END_IF;
	(* Get Status *)
	metCreate_G_NC_4 := G_NC_4.xIsCreated;	
END_IF;
END_METHOD

METHOD metCreate_H_NC_32 : BOOL

VAR

END_VAR
(* H_NC_32*)
IF NOT H_NC_32.xIsCreated THEN
	(* Ziel						UTF8->ASCII						OBJ_NAME_BASE			BacNet Text		Textlistname									BacNet Funktion																	BacNet Textlist type												TextId		*)
	H_NC_32._sObjectName		:=	fcUtfToAscii(Standard.CONCAT(	OBJ_NAME_BASE		,	fcGetBcText(	GVL_BACNET.fbBacNetParameter.metGetTextListName(enTypeOfBacNetFunktionIn := enTypeOfBacNetFunktion.Type_Automationsstation,		enTypeOfBacNetTextListIn := enTypeOfBacNetTextList.ENDING		),	'H_NC_32')));
	H_NC_32._sDescription	:= 	fcUtfToAscii(Standard.CONCAT(	OBJ_NAME_DESCRIPTION,	fcGetBcText(	GVL_BACNET.fbBacNetParameter.metGetTextListName(enTypeOfBacNetFunktionIn := enTypeOfBacNetFunktion.Type_Automationsstation,		enTypeOfBacNetTextListIn := enTypeOfBacNetTextList.DESCRIPTION	),	'H_NC_32')));
	(* Create Id from Base Id and Object Nr (Last nummber of Name *)	
	H_NC_32.Create(diInstance := 32);
	(* Check if Created *)
	IF H_NC_32.xIsCreated THEN
		(* Set Group *)
		H_NC_32.setPropertyGroup(WagoTypesBacNet.eBACnetPropertyIdentifier.PROP_DESCRIPTION							,WagoTypesBacNet.eBACnetPropertyUpdateGroup.GROUP_CYCLIC);
		
		(* Set Ack Req *)
		H_NC_32.IAckRequired.xToOffNormal	:= FALSE;
		H_NC_32.IAckRequired.xToFault		:= FALSE;
		H_NC_32.IAckRequired.xToNormal		:= FALSE;
		
		(* Ziel												UTF8->ASCII		BacNet Text		Textlistname									BacNet Funktion																	BacNet Textlist type												TextId		*)
		H_NC_32.IEventMessageTextsConfig.sToOffNormal	:=	fcUtfToAscii(	fcGetBcText(	GVL_BACNET.fbBacNetParameter.metGetTextListName(enTypeOfBacNetFunktionIn := enTypeOfBacNetFunktion.Type_Automationsstation,		enTypeOfBacNetTextListIn := enTypeOfBacNetTextList.EVENTMESSAGE	),	'H_NC_32_ToOffNormal'	));		
		H_NC_32.IEventMessageTextsConfig.sToFault		:=	fcUtfToAscii(	fcGetBcText(	GVL_BACNET.fbBacNetParameter.metGetTextListName(enTypeOfBacNetFunktionIn := enTypeOfBacNetFunktion.Type_Automationsstation,		enTypeOfBacNetTextListIn := enTypeOfBacNetTextList.EVENTMESSAGE	),	'H_NC_32_ToFault'		));		
		H_NC_32.IEventMessageTextsConfig.sToNormal		:=	fcUtfToAscii(	fcGetBcText(	GVL_BACNET.fbBacNetParameter.metGetTextListName(enTypeOfBacNetFunktionIn := enTypeOfBacNetFunktion.Type_Automationsstation,		enTypeOfBacNetTextListIn := enTypeOfBacNetTextList.EVENTMESSAGE	),	'H_NC_32_ToNormal'		));		
		
		(* Notification Class & Type *)
		H_NC_32.udiNotificationClass					:=  32;	
		H_NC_32.eNotifyType								:= 	WagoTypesBACnet.eBACnetNotifyType.NOTIFY_TYPE_ALARM;
		(* Ziel												Convert			BacNet Text		Textlistname									BacNet Funktion																	BacNet Textlist type												TextId		*)	
		H_NC_32.IPriority.usiToOffNormal				:= 	TO_USINT(fcUtfToAscii(	fcGetBcText(	GVL_BACNET.fbBacNetParameter.metGetTextListName(enTypeOfBacNetFunktionIn := enTypeOfBacNetFunktion.Type_Automationsstation,		enTypeOfBacNetTextListIn := enTypeOfBacNetTextList.NC	),	'H_NC_32_Prio_ToOffNormal'	)));	
		H_NC_32.IPriority.usiToFault					:= 	TO_USINT(fcUtfToAscii(	fcGetBcText(	GVL_BACNET.fbBacNetParameter.metGetTextListName(enTypeOfBacNetFunktionIn := enTypeOfBacNetFunktion.Type_Automationsstation,		enTypeOfBacNetTextListIn := enTypeOfBacNetTextList.NC	),	'H_NC_32_Prio_ToFault'		)));	
		H_NC_32.IPriority.usiToNormal					:= 	TO_USINT(fcUtfToAscii(	fcGetBcText(	GVL_BACNET.fbBacNetParameter.metGetTextListName(enTypeOfBacNetFunktionIn := enTypeOfBacNetFunktion.Type_Automationsstation,		enTypeOfBacNetTextListIn := enTypeOfBacNetTextList.NC	),	'H_NC_32_Prio_ToNormal'		)));	
		
	ELSE
		H_NC_32.Delete();
	END_IF;
	(* Get Status *)
	metCreate_H_NC_32 := H_NC_32.xIsCreated;	
END_IF;
END_METHOD

METHOD metCreate_H_NC_33 : BOOL

VAR

END_VAR
(* H_NC_33*)
IF NOT H_NC_33.xIsCreated THEN
	(* Ziel						UTF8->ASCII						OBJ_NAME_BASE			BacNet Text		Textlistname									BacNet Funktion																	BacNet Textlist type												TextId		*)
	H_NC_33._sObjectName		:=	fcUtfToAscii(Standard.CONCAT(	OBJ_NAME_BASE		,	fcGetBcText(	GVL_BACNET.fbBacNetParameter.metGetTextListName(enTypeOfBacNetFunktionIn := enTypeOfBacNetFunktion.Type_Automationsstation,		enTypeOfBacNetTextListIn := enTypeOfBacNetTextList.ENDING		),	'H_NC_33')));
	H_NC_33._sDescription	:= 	fcUtfToAscii(Standard.CONCAT(	OBJ_NAME_DESCRIPTION,	fcGetBcText(	GVL_BACNET.fbBacNetParameter.metGetTextListName(enTypeOfBacNetFunktionIn := enTypeOfBacNetFunktion.Type_Automationsstation,		enTypeOfBacNetTextListIn := enTypeOfBacNetTextList.DESCRIPTION	),	'H_NC_33')));
	(* Create Id from Base Id and Object Nr (Last nummber of Name *)	
	H_NC_33.Create(diInstance := 33);
	(* Check if Created *)
	IF H_NC_33.xIsCreated THEN
		(* Set Group *)
		H_NC_33.setPropertyGroup(WagoTypesBacNet.eBACnetPropertyIdentifier.PROP_DESCRIPTION							,WagoTypesBacNet.eBACnetPropertyUpdateGroup.GROUP_CYCLIC);
		
		(* Set Ack Req *)
		H_NC_33.IAckRequired.xToOffNormal	:= FALSE;
		H_NC_33.IAckRequired.xToFault		:= TRUE;
		H_NC_33.IAckRequired.xToNormal		:= FALSE;
		
		(* Ziel												UTF8->ASCII		BacNet Text		Textlistname									BacNet Funktion																	BacNet Textlist type												TextId		*)
		H_NC_33.IEventMessageTextsConfig.sToOffNormal	:=	fcUtfToAscii(	fcGetBcText(	GVL_BACNET.fbBacNetParameter.metGetTextListName(enTypeOfBacNetFunktionIn := enTypeOfBacNetFunktion.Type_Automationsstation,		enTypeOfBacNetTextListIn := enTypeOfBacNetTextList.EVENTMESSAGE	),	'H_NC_33_ToOffNormal'	));		
		H_NC_33.IEventMessageTextsConfig.sToFault		:=	fcUtfToAscii(	fcGetBcText(	GVL_BACNET.fbBacNetParameter.metGetTextListName(enTypeOfBacNetFunktionIn := enTypeOfBacNetFunktion.Type_Automationsstation,		enTypeOfBacNetTextListIn := enTypeOfBacNetTextList.EVENTMESSAGE	),	'H_NC_33_ToFault'		));		
		H_NC_33.IEventMessageTextsConfig.sToNormal		:=	fcUtfToAscii(	fcGetBcText(	GVL_BACNET.fbBacNetParameter.metGetTextListName(enTypeOfBacNetFunktionIn := enTypeOfBacNetFunktion.Type_Automationsstation,		enTypeOfBacNetTextListIn := enTypeOfBacNetTextList.EVENTMESSAGE	),	'H_NC_33_ToNormal'		));		
		
		(* Notification Class & Type *)
		H_NC_33.udiNotificationClass					:=  33;	
		H_NC_33.eNotifyType								:= 	WagoTypesBACnet.eBACnetNotifyType.NOTIFY_TYPE_ALARM;
		(* Ziel												Convert			BacNet Text		Textlistname									BacNet Funktion																	BacNet Textlist type												TextId		*)	
		H_NC_33.IPriority.usiToOffNormal				:= 	TO_USINT(fcUtfToAscii(	fcGetBcText(	GVL_BACNET.fbBacNetParameter.metGetTextListName(enTypeOfBacNetFunktionIn := enTypeOfBacNetFunktion.Type_Automationsstation,		enTypeOfBacNetTextListIn := enTypeOfBacNetTextList.NC	),	'H_NC_33_Prio_ToOffNormal'	)));	
		H_NC_33.IPriority.usiToFault					:= 	TO_USINT(fcUtfToAscii(	fcGetBcText(	GVL_BACNET.fbBacNetParameter.metGetTextListName(enTypeOfBacNetFunktionIn := enTypeOfBacNetFunktion.Type_Automationsstation,		enTypeOfBacNetTextListIn := enTypeOfBacNetTextList.NC	),	'H_NC_33_Prio_ToFault'		)));	
		H_NC_33.IPriority.usiToNormal					:= 	TO_USINT(fcUtfToAscii(	fcGetBcText(	GVL_BACNET.fbBacNetParameter.metGetTextListName(enTypeOfBacNetFunktionIn := enTypeOfBacNetFunktion.Type_Automationsstation,		enTypeOfBacNetTextListIn := enTypeOfBacNetTextList.NC	),	'H_NC_33_Prio_ToNormal'		)));	
		
	ELSE
		H_NC_33.Delete();
	END_IF;
	(* Get Status *)
	metCreate_H_NC_33 := H_NC_33.xIsCreated;	
END_IF;
END_METHOD

METHOD metCreate_H_NC_34 : BOOL

VAR

END_VAR
(* H_NC_34*)
IF NOT H_NC_34.xIsCreated THEN
	(* Ziel						UTF8->ASCII						OBJ_NAME_BASE			BacNet Text		Textlistname									BacNet Funktion																	BacNet Textlist type												TextId		*)
	H_NC_34._sObjectName		:=	fcUtfToAscii(Standard.CONCAT(	OBJ_NAME_BASE		,	fcGetBcText(	GVL_BACNET.fbBacNetParameter.metGetTextListName(enTypeOfBacNetFunktionIn := enTypeOfBacNetFunktion.Type_Automationsstation,		enTypeOfBacNetTextListIn := enTypeOfBacNetTextList.ENDING		),	'H_NC_34')));
	H_NC_34._sDescription	:= 	fcUtfToAscii(Standard.CONCAT(	OBJ_NAME_DESCRIPTION,	fcGetBcText(	GVL_BACNET.fbBacNetParameter.metGetTextListName(enTypeOfBacNetFunktionIn := enTypeOfBacNetFunktion.Type_Automationsstation,		enTypeOfBacNetTextListIn := enTypeOfBacNetTextList.DESCRIPTION	),	'H_NC_34')));
	(* Create Id from Base Id and Object Nr (Last nummber of Name *)	
	H_NC_34.Create(diInstance := 34);
	(* Check if Created *)
	IF H_NC_34.xIsCreated THEN
		(* Set Group *)
		H_NC_34.setPropertyGroup(WagoTypesBacNet.eBACnetPropertyIdentifier.PROP_DESCRIPTION							,WagoTypesBacNet.eBACnetPropertyUpdateGroup.GROUP_CYCLIC);
		
		(* Set Ack Req *)
		H_NC_34.IAckRequired.xToOffNormal	:= TRUE;
		H_NC_34.IAckRequired.xToFault		:= TRUE;
		H_NC_34.IAckRequired.xToNormal		:= FALSE;
		
		(* Ziel												UTF8->ASCII		BacNet Text		Textlistname									BacNet Funktion																	BacNet Textlist type												TextId		*)
		H_NC_34.IEventMessageTextsConfig.sToOffNormal	:=	fcUtfToAscii(	fcGetBcText(	GVL_BACNET.fbBacNetParameter.metGetTextListName(enTypeOfBacNetFunktionIn := enTypeOfBacNetFunktion.Type_Automationsstation,		enTypeOfBacNetTextListIn := enTypeOfBacNetTextList.EVENTMESSAGE	),	'H_NC_34_ToOffNormal'	));		
		H_NC_34.IEventMessageTextsConfig.sToFault		:=	fcUtfToAscii(	fcGetBcText(	GVL_BACNET.fbBacNetParameter.metGetTextListName(enTypeOfBacNetFunktionIn := enTypeOfBacNetFunktion.Type_Automationsstation,		enTypeOfBacNetTextListIn := enTypeOfBacNetTextList.EVENTMESSAGE	),	'H_NC_34_ToFault'		));		
		H_NC_34.IEventMessageTextsConfig.sToNormal		:=	fcUtfToAscii(	fcGetBcText(	GVL_BACNET.fbBacNetParameter.metGetTextListName(enTypeOfBacNetFunktionIn := enTypeOfBacNetFunktion.Type_Automationsstation,		enTypeOfBacNetTextListIn := enTypeOfBacNetTextList.EVENTMESSAGE	),	'H_NC_34_ToNormal'		));		
		
		(* Notification Class & Type *)
		H_NC_34.udiNotificationClass					:=  34;	
		H_NC_34.eNotifyType								:= 	WagoTypesBACnet.eBACnetNotifyType.NOTIFY_TYPE_ALARM;
		(* Ziel												Convert			BacNet Text		Textlistname									BacNet Funktion																	BacNet Textlist type												TextId		*)	
		H_NC_34.IPriority.usiToOffNormal				:= 	TO_USINT(fcUtfToAscii(	fcGetBcText(	GVL_BACNET.fbBacNetParameter.metGetTextListName(enTypeOfBacNetFunktionIn := enTypeOfBacNetFunktion.Type_Automationsstation,		enTypeOfBacNetTextListIn := enTypeOfBacNetTextList.NC	),	'H_NC_34_Prio_ToOffNormal'	)));	
		H_NC_34.IPriority.usiToFault					:= 	TO_USINT(fcUtfToAscii(	fcGetBcText(	GVL_BACNET.fbBacNetParameter.metGetTextListName(enTypeOfBacNetFunktionIn := enTypeOfBacNetFunktion.Type_Automationsstation,		enTypeOfBacNetTextListIn := enTypeOfBacNetTextList.NC	),	'H_NC_34_Prio_ToFault'		)));	
		H_NC_34.IPriority.usiToNormal					:= 	TO_USINT(fcUtfToAscii(	fcGetBcText(	GVL_BACNET.fbBacNetParameter.metGetTextListName(enTypeOfBacNetFunktionIn := enTypeOfBacNetFunktion.Type_Automationsstation,		enTypeOfBacNetTextListIn := enTypeOfBacNetTextList.NC	),	'H_NC_34_Prio_ToNormal'		)));	
		
	ELSE
		H_NC_34.Delete();
	END_IF;
	(* Get Status *)
	metCreate_H_NC_34 := H_NC_34.xIsCreated;	
END_IF;
END_METHOD

METHOD metCreate_I_NC_65 : BOOL

VAR

END_VAR
(* I_NC_65*)
IF NOT I_NC_65.xIsCreated THEN
	(* Ziel						UTF8->ASCII						OBJ_NAME_BASE			BacNet Text		Textlistname									BacNet Funktion																	BacNet Textlist type												TextId		*)
	I_NC_65._sObjectName		:=	fcUtfToAscii(Standard.CONCAT(	OBJ_NAME_BASE		,	fcGetBcText(	GVL_BACNET.fbBacNetParameter.metGetTextListName(enTypeOfBacNetFunktionIn := enTypeOfBacNetFunktion.Type_Automationsstation,		enTypeOfBacNetTextListIn := enTypeOfBacNetTextList.ENDING		),	'I_NC_65')));
	I_NC_65._sDescription	:= 	fcUtfToAscii(Standard.CONCAT(	OBJ_NAME_DESCRIPTION,	fcGetBcText(	GVL_BACNET.fbBacNetParameter.metGetTextListName(enTypeOfBacNetFunktionIn := enTypeOfBacNetFunktion.Type_Automationsstation,		enTypeOfBacNetTextListIn := enTypeOfBacNetTextList.DESCRIPTION	),	'I_NC_65')));
	(* Create Id from Base Id and Object Nr (Last nummber of Name *)	
	I_NC_65.Create(diInstance := 65);
	(* Check if Created *)
	IF I_NC_65.xIsCreated THEN
		(* Set Group *)
		I_NC_65.setPropertyGroup(WagoTypesBacNet.eBACnetPropertyIdentifier.PROP_DESCRIPTION							,WagoTypesBacNet.eBACnetPropertyUpdateGroup.GROUP_CYCLIC);
		
		(* Set Ack Req *)
		I_NC_65.IAckRequired.xToOffNormal	:= FALSE;
		I_NC_65.IAckRequired.xToFault		:= TRUE;
		I_NC_65.IAckRequired.xToNormal		:= FALSE;
		
		(* Ziel												UTF8->ASCII		BacNet Text		Textlistname									BacNet Funktion																	BacNet Textlist type												TextId		*)
		I_NC_65.IEventMessageTextsConfig.sToOffNormal	:=	fcUtfToAscii(	fcGetBcText(	GVL_BACNET.fbBacNetParameter.metGetTextListName(enTypeOfBacNetFunktionIn := enTypeOfBacNetFunktion.Type_Automationsstation,		enTypeOfBacNetTextListIn := enTypeOfBacNetTextList.EVENTMESSAGE	),	'I_NC_65_ToOffNormal'	));		
		I_NC_65.IEventMessageTextsConfig.sToFault		:=	fcUtfToAscii(	fcGetBcText(	GVL_BACNET.fbBacNetParameter.metGetTextListName(enTypeOfBacNetFunktionIn := enTypeOfBacNetFunktion.Type_Automationsstation,		enTypeOfBacNetTextListIn := enTypeOfBacNetTextList.EVENTMESSAGE	),	'I_NC_65_ToFault'		));		
		I_NC_65.IEventMessageTextsConfig.sToNormal		:=	fcUtfToAscii(	fcGetBcText(	GVL_BACNET.fbBacNetParameter.metGetTextListName(enTypeOfBacNetFunktionIn := enTypeOfBacNetFunktion.Type_Automationsstation,		enTypeOfBacNetTextListIn := enTypeOfBacNetTextList.EVENTMESSAGE	),	'I_NC_65_ToNormal'		));		
		
		(* Notification Class & Type *)
		I_NC_65.udiNotificationClass					:=  65;	
		I_NC_65.eNotifyType								:= 	WagoTypesBACnet.eBACnetNotifyType.NOTIFY_TYPE_ALARM;
		(* Ziel												Convert			BacNet Text		Textlistname									BacNet Funktion																	BacNet Textlist type												TextId		*)	
		I_NC_65.IPriority.usiToOffNormal				:= 	TO_USINT(fcUtfToAscii(	fcGetBcText(	GVL_BACNET.fbBacNetParameter.metGetTextListName(enTypeOfBacNetFunktionIn := enTypeOfBacNetFunktion.Type_Automationsstation,		enTypeOfBacNetTextListIn := enTypeOfBacNetTextList.NC	),	'I_NC_65_Prio_ToOffNormal'	)));	
		I_NC_65.IPriority.usiToFault					:= 	TO_USINT(fcUtfToAscii(	fcGetBcText(	GVL_BACNET.fbBacNetParameter.metGetTextListName(enTypeOfBacNetFunktionIn := enTypeOfBacNetFunktion.Type_Automationsstation,		enTypeOfBacNetTextListIn := enTypeOfBacNetTextList.NC	),	'I_NC_65_Prio_ToFault'		)));	
		I_NC_65.IPriority.usiToNormal					:= 	TO_USINT(fcUtfToAscii(	fcGetBcText(	GVL_BACNET.fbBacNetParameter.metGetTextListName(enTypeOfBacNetFunktionIn := enTypeOfBacNetFunktion.Type_Automationsstation,		enTypeOfBacNetTextListIn := enTypeOfBacNetTextList.NC	),	'I_NC_65_Prio_ToNormal'		)));	
		
	ELSE
		I_NC_65.Delete();
	END_IF;
	(* Get Status *)
	metCreate_I_NC_65 := I_NC_65.xIsCreated;	
END_IF;
END_METHOD

END_FUNCTION_BLOCK

// 30 Program Organization Units/FCs/XMLFcs/XML BacNet Override/DEVICE/fcXMLDeviceOverride
FUNCTION fcXMLDeviceOverride : BOOL
VAR_INPUT
	I_BACnetDevice_small				:	WagoTypesBacnet.I_BACnetDevice_small;
	diNewObjId							:	DINT;
	stNewObjName						:	STRING(64);
END_VAR
VAR
	stBacNetDeviceId					:	STRING[8];
	stBacNetDeviceIdNew					:	STRING[8];
	stParentPath						:	STRING[80];
	stXmlPath							:	STRING[80];
END_VAR

IF __QUERYINTERFACE(I_BACnetDevice_small,I_BACnetDevice_small) THEN
	// Get Information
	stBacNetDeviceId 		:= fcBacNetIdToIdWitType(I_BACnetDevice_small.IObjectIdentifier.diInstance,I_BACnetDevice_small.IObjectIdentifier.eObjectType);
	stBacNetDeviceIdNew		:= fcBacNetIdToIdWitType(diNewObjId,I_BACnetDevice_small.IObjectIdentifier.eObjectType);
	GVL_BACNET.stBacNetDeviceId := stBacNetDeviceIdNew;
	// xml path
	stXmlPath := '/home/user/bacnet/config/override.xml';
	// Create BacNet Object 
	stParentPath := '';
	stParentPath := '//*/objLst';
	IF fcXMLCheckNode(stParentPath,'obj','id',stBacNetDeviceId,'','',stXmlPath) THEN
		IF fcXMLUpdateAttribute(stParentPath,'obj','id',stBacNetDeviceId,'id',stBacNetDeviceIdNew,stXmlPath) THEN	
			fcXMLDeviceOverride := TRUE;
		END_IF;
		// Create PROP_OBJECT_NAME
		stParentPath := '';
		stParentPath := CONCAT('//*/objLst/obj[@id=$'',CONCAT(stBacNetDeviceIdNew,'$']'));	
		IF fcXMLAddNode(stParentPath,'p','id',TO_STRING(TO_INT(WagoTypesBACnet.eBACnetPropertyIdentifier.PROP_OBJECT_NAME)),'','',stXmlPath,FALSE) THEN	
			fcXMLDeviceOverride := TRUE;
		END_IF;
			// Create Node PROP_OBJECT_NAME
			stParentPath := '';
			stParentPath := CONCAT(CONCAT(CONCAT(CONCAT('//*/objLst/obj[@id=$'',stBacNetDeviceIdNew),'$']/p[@id=$''),TO_STRING(TO_INT(WagoTypesBACnet.eBACnetPropertyIdentifier.PROP_OBJECT_NAME))),'$']');	
			IF fcXMLCheckNode(stParentPath,'n','t','112','','',stXmlPath) THEN
				fcXMLUpdateAttribute(stParentPath,'n','t','112','v',stNewObjName,stXmlPath);
				fcXMLDeviceOverride := TRUE;
			ELSE
				IF fcXMLAddNode(stParentPath,'n','t','112','v',stNewObjName,stXmlPath,FALSE) THEN	
					fcXMLDeviceOverride := TRUE;
				END_IF;
			END_IF;
		// Create PROP_OBJECT_IDENTIFIER
		stParentPath := '';
		stParentPath := CONCAT('//*/objLst/obj[@id=$'',CONCAT(stBacNetDeviceIdNew,'$']'));	
		IF fcXMLAddNode(stParentPath,'p','id',TO_STRING(TO_INT(WagoTypesBACnet.eBACnetPropertyIdentifier.PROP_OBJECT_IDENTIFIER)),'','',stXmlPath,FALSE) THEN	
			fcXMLDeviceOverride := TRUE;
		END_IF;
			// Create Node PROP_OBJECT_IDENTIFIER
			stParentPath := '';
			stParentPath := CONCAT(CONCAT(CONCAT(CONCAT('//*/objLst/obj[@id=$'',stBacNetDeviceIdNew),'$']/p[@id=$''),TO_STRING(TO_INT(WagoTypesBACnet.eBACnetPropertyIdentifier.PROP_OBJECT_IDENTIFIER))),'$']');	
			IF fcXMLCheckNode(stParentPath,'n','t','192','','',stXmlPath) THEN
				IF fcXMLUpdateAttribute(stParentPath,'n','t','192','v',stBacNetDeviceIdNew,stXmlPath) THEN
					fcXMLDeviceOverride := TRUE;
				END_IF;
			ELSE
				IF fcXMLAddNode(stParentPath,'n','t','192','v',stBacNetDeviceIdNew,stXmlPath,FALSE) THEN	
					fcXMLDeviceOverride := TRUE;
				END_IF;
			END_IF;
	END_IF;
END_IF;

END_FUNCTION

// 30 Program Organization Units/FBs/AT_FUNKTIONEN/AT_ANLAGEFUNKTION/FB_AT_ANLAGEFUNKTION
FUNCTION_BLOCK FB_AT_ANLAGEFUNKTION EXTENDS FB_OBJ_ID_BASE
VAR_INPUT
	xObjektSchutz		:	BOOL;
	xTechnischerAlarm	:	BOOL;
	xTechnischeStörung	:	BOOL;
	xWartungsmeldung	:	BOOL;
	xBedienungLokal		:	BOOL;
	xAlarmUnterdrückung	:	BOOL;
	xAcknowledge		:	BOOL;
END_VAR
VAR_OUTPUT
	xZeitschaltUhr		:	BOOL;
END_VAR
VAR
	(* BacNet Objects *)
	A_BV_1				:	WagoSysBACnet.FbBinaryValue_large(-1);					// Sammelmeldung Objektschutz
	B_BV_2				:	WagoSysBACnet.FbBinaryValue_large(-1);					// Sammelmeldung Technischer Alarm
	C_BV_3				:	WagoSysBACnet.FbBinaryValue_large(-1);					// Sammelmeldung Technische Störung
	D_BV_4				:	WagoSysBACnet.FbBinaryValue_large(-1);					// Sammelmeldung Wartungsmeldung
	E_BI_1				:	WagoSysBACnet.FbBinaryInput_large(-1);					// Bedienung Lokal
	F_BV_5				:	WagoSysBACnet.FbBinaryValue_large(-1);					// Alarmunterdrückung
	G_BO_1				:	WagoSysBACnet.FbBinaryOutput_large(-1);					// Signalisation Betrieb
	H_BO_2				:	WagoSysBACnet.FbBinaryOutput_large(-1);					// Signalisation Sammelalarm
	I_BO_3				:	WagoSysBACnet.FbBinaryOutput_large(-1);					// Signalisation Bedienung Lokal
	J_SC_1				:	WagoSysBACnet.FbSchedule_large(-1);						// Zeitschaltuhr
END_VAR
VAR CONSTANT
	usiAnzBacNetObj	:	USINT	:= 10;
END_VAR

(* Call Base FB*)
SUPER^();
(* Cyclic Action *)
IF xCreatet THEN
	(* DESCTIPTION FIX *)
	metCYCLIC_DESCRIPTION_FIX();
	(* Get Revision *)
	CASE GVL_BACNET.fbBacNetParameter.proKBOB_REV OF
		(* KBOB 2021 V2 *)
		enKBOB_REV.KBOB_REV2021_V2:
			metCYCLIC_KBOB_2021_V2();
		(* KBOB 2017 V1 *)
		enKBOB_REV.KBOB_REV2017_V1:
			metCYCLIC_KBOB_2017_V1();
		(* Default *)
		ELSE
			metCYCLIC_KBOB_2021_V2();
	END_CASE;	
END_IF;

METHOD metCREATE_STRUCTVIEW_KBOB_2021_V2 : BOOL
VAR_INPUT
END_VAR
CASE usiCreateCase OF
	1:
		fcXMLStructuredView(THIS^,A_BV_1.IObjectIdentifier);
	2:
		fcXMLStructuredView(THIS^,B_BV_2.IObjectIdentifier);
	3:
		fcXMLStructuredView(THIS^,C_BV_3.IObjectIdentifier);
	4:
		fcXMLStructuredView(THIS^,D_BV_4.IObjectIdentifier);
	5:
		fcXMLStructuredView(THIS^,E_BI_1.IObjectIdentifier);
	6:
		fcXMLStructuredView(THIS^,F_BV_5.IObjectIdentifier);
	7:
		fcXMLStructuredView(THIS^,G_BO_1.IObjectIdentifier);
	8:
		fcXMLStructuredView(THIS^,H_BO_2.IObjectIdentifier);
	9:
		fcXMLStructuredView(THIS^,I_BO_3.IObjectIdentifier);
	10:
		fcXMLStructuredView(THIS^,J_SC_1.IObjectIdentifier);
		fcXMLAddStructuredViewToDevice(THIS^);	
	0: 
		usiCreateCase := 1;
ELSE
	usiCreateCase := 0;
END_CASE
END_METHOD

METHOD metCREATE_KBOB_2021_V2 : BOOL;
VAR_INPUT
END_VAR
VAR
	oStatus		:	WagoSysErrorBase.FbResult;
	usiErrors	:	USINT;
END_VAR
(* Resett *)
usiErrors := 0;	

(* Create Objeccts *)
CASE usiCreateCase OF
	1:	
		usiErrors := usiErrors + TO_USINT(NOT metCreate_A_BV_1());
	2:
		usiErrors := usiErrors + TO_USINT(NOT metCreate_B_BV_2());
	3:	
		usiErrors := usiErrors + TO_USINT(NOT metCreate_C_BV_3());
	4:	
		usiErrors := usiErrors + TO_USINT(NOT metCreate_D_BV_4());
	5:
		usiErrors := usiErrors + TO_USINT(NOT metCreate_E_BI_1());
	6:	
		usiErrors := usiErrors + TO_USINT(NOT metCreate_F_BV_5());
	7:
		usiErrors := usiErrors + TO_USINT(NOT metCreate_G_BO_1());
	8:	
		usiErrors := usiErrors + TO_USINT(NOT metCreate_H_BO_2());
	9:
		usiErrors := usiErrors + TO_USINT(NOT metCreate_I_BO_3());
	10:
		usiErrors := usiErrors + TO_USINT(NOT metCreate_J_SC_1());
	0: 
		usiCreateCase := 1;
ELSE
	usiCreateCase := 0;
END_CASE;

(* STRUCT VIEW *)
metCREATE_STRUCTVIEW_KBOB_2021_V2();

(* OK = 0*)
metCREATE_KBOB_2021_V2 := NOT TO_BOOL(usiErrors);
END_METHOD

METHOD metCreate_H_BO_2 : BOOL
(* H_BO_2*)
IF NOT H_BO_2.xIsCreated THEN
	(* Ziel						UTF8->ASCII						OBJ_NAME_BASE			BacNet Text		Textlistname									BacNet Funktion																BacNet Textlist type												TextId		*)
	H_BO_2._sObjectName		:=	fcUtfToAscii(Standard.CONCAT(	OBJ_NAME_BASE		,	fcGetBcText(	GVL_BACNET.fbBacNetParameter.metGetTextListName(enTypeOfBacNetFunktionIn := enTypeOfBacNetFunktion.Type_Anlagefunktion,		enTypeOfBacNetTextListIn := enTypeOfBacNetTextList.ENDING		),	'H_BO_2')));
	H_BO_2._sDescription	:= 	fcUtfToAscii(Standard.CONCAT(	OBJ_NAME_DESCRIPTION,	fcGetBcText(	GVL_BACNET.fbBacNetParameter.metGetTextListName(enTypeOfBacNetFunktionIn := enTypeOfBacNetFunktion.Type_Anlagefunktion,		enTypeOfBacNetTextListIn := enTypeOfBacNetTextList.DESCRIPTION	),	'H_BO_2')));
	(* Create Id from Base Id and Object Nr (Last nummber of Name *)	
	H_BO_2.Create(diInstance := TO_DINT(Standard.CONCAT(TO_STRING(dwOBJ_ID_BASE),'1')));
	(* Check if Created *)
	IF H_BO_2.xIsCreated THEN
		(* Set Group *)
		H_BO_2.setPropertyGroup(WagoTypesBacNet.eBACnetPropertyIdentifier.PROP_PRESENT_VALUE						,WagoTypesBacNet.eBACnetPropertyUpdateGroup.GROUP_CYCLIC);
		H_BO_2.setPropertyGroup(WagoTypesBacNet.eBACnetPropertyIdentifier.PROP_PRIORITY_ARRAY						,WagoTypesBacNet.eBACnetPropertyUpdateGroup.GROUP_CYCLIC);
		H_BO_2.setPropertyGroup(WagoTypesBacNet.eBACnetPropertyIdentifier.PROP_ELAPSED_ACTIVE_TIME					,WagoTypesBacNet.eBACnetPropertyUpdateGroup.GROUP_CYCLIC);
		H_BO_2.setPropertyGroup(WagoTypesBacNet.eBACnetPropertyIdentifier.PROP_DESCRIPTION							,WagoTypesBacNet.eBACnetPropertyUpdateGroup.GROUP_CYCLIC);
		H_BO_2.setPropertyGroup(WagoTypesBacNet.eBACnetPropertyIdentifier.PROP_EVENT_MESSAGE_TEXTS_CONFIG			,WagoTypesBacNet.eBACnetPropertyUpdateGroup.GROUP_CYCLIC);
			
		(* Ziel												UTF8->ASCII		BacNet Text		Textlistname									BacNet Funktion																BacNet Textlist type												TextId		*)
		H_BO_2.IEventMessageTextsConfig.sToOffNormal	:=	fcUtfToAscii(	fcGetBcText(	GVL_BACNET.fbBacNetParameter.metGetTextListName(enTypeOfBacNetFunktionIn := enTypeOfBacNetFunktion.Type_Anlagefunktion,		enTypeOfBacNetTextListIn := enTypeOfBacNetTextList.EVENTMESSAGE	),	'H_BO_2_ToOffNormal'	));		
		H_BO_2.IEventMessageTextsConfig.sToFault		:=	fcUtfToAscii(	fcGetBcText(	GVL_BACNET.fbBacNetParameter.metGetTextListName(enTypeOfBacNetFunktionIn := enTypeOfBacNetFunktion.Type_Anlagefunktion,		enTypeOfBacNetTextListIn := enTypeOfBacNetTextList.EVENTMESSAGE	),	'H_BO_2_ToFault'		));		
		H_BO_2.IEventMessageTextsConfig.sToNormal		:=	fcUtfToAscii(	fcGetBcText(	GVL_BACNET.fbBacNetParameter.metGetTextListName(enTypeOfBacNetFunktionIn := enTypeOfBacNetFunktion.Type_Anlagefunktion,		enTypeOfBacNetTextListIn := enTypeOfBacNetTextList.EVENTMESSAGE	),	'H_BO_2_ToNormal'		));		

		(* Ziel												UTF8->ASCII		BacNet Text		Textlistname									BacNet Funktion																BacNet Textlist type												TextId		*)	
		H_BO_2.sActiveText								:= 	fcUtfToAscii(	fcGetBcText(	GVL_BACNET.fbBacNetParameter.metGetTextListName(enTypeOfBacNetFunktionIn := enTypeOfBacNetFunktion.Type_Anlagefunktion,		enTypeOfBacNetTextListIn := enTypeOfBacNetTextList.PRESENTVALUE	),	'H_BO_2_ST_ACTIVE'		));
		H_BO_2.sInactiveText							:= 	fcUtfToAscii(	fcGetBcText(	GVL_BACNET.fbBacNetParameter.metGetTextListName(enTypeOfBacNetFunktionIn := enTypeOfBacNetFunktion.Type_Anlagefunktion,		enTypeOfBacNetTextListIn := enTypeOfBacNetTextList.PRESENTVALUE	),	'H_BO_2_ST_INACTIVE'	));	

		(* Ziel												Convert			BacNet Text		Textlistname									BacNet Funktion																BacNet Textlist type												TextId		*)	
		H_BO_2.udiNotificationClass						:= 	TO_UDINT	(	fcGetBcText(	GVL_BACNET.fbBacNetParameter.metGetTextListName(enTypeOfBacNetFunktionIn := enTypeOfBacNetFunktion.Type_Anlagefunktion,		enTypeOfBacNetTextListIn := enTypeOfBacNetTextList.NC			),	'H_BO_2_NC'	));	
		H_BO_2.eNotifyType								:= 	WagoTypesBACnet.eBACnetNotifyType.NOTIFY_TYPE_ALARM;
		
	ELSE
		H_BO_2.Delete();
	END_IF;
	(* Get Status *)
	metCreate_H_BO_2 := H_BO_2.xIsCreated;	
END_IF;
END_METHOD

METHOD metCreate_I_BO_3 : BOOL
(* I_BO_3*)
IF NOT I_BO_3.xIsCreated THEN
	(* Ziel						UTF8->ASCII						OBJ_NAME_BASE			BacNet Text		Textlistname									BacNet Funktion																BacNet Textlist type												TextId		*)
	I_BO_3._sObjectName		:=	fcUtfToAscii(Standard.CONCAT(	OBJ_NAME_BASE		,	fcGetBcText(	GVL_BACNET.fbBacNetParameter.metGetTextListName(enTypeOfBacNetFunktionIn := enTypeOfBacNetFunktion.Type_Anlagefunktion,		enTypeOfBacNetTextListIn := enTypeOfBacNetTextList.ENDING		),	'I_BO_3')));
	I_BO_3._sDescription	:= 	fcUtfToAscii(Standard.CONCAT(	OBJ_NAME_DESCRIPTION,	fcGetBcText(	GVL_BACNET.fbBacNetParameter.metGetTextListName(enTypeOfBacNetFunktionIn := enTypeOfBacNetFunktion.Type_Anlagefunktion,		enTypeOfBacNetTextListIn := enTypeOfBacNetTextList.DESCRIPTION	),	'I_BO_3')));
	(* Create Id from Base Id and Object Nr (Last nummber of Name *)	
	I_BO_3.Create(diInstance := TO_DINT(Standard.CONCAT(TO_STRING(dwOBJ_ID_BASE),'1')));
	(* Check if Created *)
	IF I_BO_3.xIsCreated THEN
		(* Set Group *)
		I_BO_3.setPropertyGroup(WagoTypesBacNet.eBACnetPropertyIdentifier.PROP_PRESENT_VALUE						,WagoTypesBacNet.eBACnetPropertyUpdateGroup.GROUP_CYCLIC);
		I_BO_3.setPropertyGroup(WagoTypesBacNet.eBACnetPropertyIdentifier.PROP_PRIORITY_ARRAY						,WagoTypesBacNet.eBACnetPropertyUpdateGroup.GROUP_CYCLIC);
		I_BO_3.setPropertyGroup(WagoTypesBacNet.eBACnetPropertyIdentifier.PROP_ELAPSED_ACTIVE_TIME					,WagoTypesBacNet.eBACnetPropertyUpdateGroup.GROUP_CYCLIC);
		I_BO_3.setPropertyGroup(WagoTypesBacNet.eBACnetPropertyIdentifier.PROP_DESCRIPTION							,WagoTypesBacNet.eBACnetPropertyUpdateGroup.GROUP_CYCLIC);
		I_BO_3.setPropertyGroup(WagoTypesBacNet.eBACnetPropertyIdentifier.PROP_EVENT_MESSAGE_TEXTS_CONFIG			,WagoTypesBacNet.eBACnetPropertyUpdateGroup.GROUP_CYCLIC);
			
		(* Ziel												UTF8->ASCII		BacNet Text		Textlistname									BacNet Funktion																BacNet Textlist type												TextId		*)
		I_BO_3.IEventMessageTextsConfig.sToOffNormal	:=	fcUtfToAscii(	fcGetBcText(	GVL_BACNET.fbBacNetParameter.metGetTextListName(enTypeOfBacNetFunktionIn := enTypeOfBacNetFunktion.Type_Anlagefunktion,		enTypeOfBacNetTextListIn := enTypeOfBacNetTextList.EVENTMESSAGE	),	'I_BO_3_ToOffNormal'	));		
		I_BO_3.IEventMessageTextsConfig.sToFault		:=	fcUtfToAscii(	fcGetBcText(	GVL_BACNET.fbBacNetParameter.metGetTextListName(enTypeOfBacNetFunktionIn := enTypeOfBacNetFunktion.Type_Anlagefunktion,		enTypeOfBacNetTextListIn := enTypeOfBacNetTextList.EVENTMESSAGE	),	'I_BO_3_ToFault'		));		
		I_BO_3.IEventMessageTextsConfig.sToNormal		:=	fcUtfToAscii(	fcGetBcText(	GVL_BACNET.fbBacNetParameter.metGetTextListName(enTypeOfBacNetFunktionIn := enTypeOfBacNetFunktion.Type_Anlagefunktion,		enTypeOfBacNetTextListIn := enTypeOfBacNetTextList.EVENTMESSAGE	),	'I_BO_3_ToNormal'		));		

